DATA_BLOCK "DB09_TablePos"   // DB9
{ S7_Optimized_Access := 'FALSE' }
AUTHOR : Robopac
VERSION : 0.0
// stored: AutoNumber false, IsOnlyStoredInLoadMemory false, IsWriteProtectedInAS false
   VAR RETAIN
      dbx0_0 : Bool := FALSE;
      dbx0_1 : Bool := FALSE;
      dbx0_2 : Bool := TRUE;
      dbx0_3 : Bool := FALSE;
      dbx0_4 : Bool := FALSE;
      dbx0_5 : Bool := FALSE;
      dbx0_6 : Bool := FALSE;
      dbx0_7 : Bool := FALSE;
      dbx1_0 : Bool := FALSE;   // Table rotation axis movement forward
      dbx1_1 : Bool := FALSE;   // Table rotation axis movement backward
      dbx1_2 : Bool := FALSE;   // Table rotation axis movement inside low speed area
      dbx1_3 : Bool := FALSE;   // Table rotation axis movement low speed
      dbx1_4 : Bool := FALSE;   // Table rotation forward
      dbx1_5 : Bool := FALSE;   // Table rotation backward
      dbx1_6 : Bool := TRUE;
      dbx1_7 : Bool := FALSE;
      dbx2_0 : Bool := FALSE;
      dbx2_1 : Bool := FALSE;
      dbx2_2 : Bool := FALSE;
      dbx2_3 : Bool := FALSE;
      dbx2_4 : Bool := FALSE;
      dbx2_5 : Bool := FALSE;
      dbx2_6 : Bool := FALSE;
      dbx2_7 : Bool := FALSE;
      dbx3_0 : Bool := FALSE;   // Table rotation: Support for encoder running control
      dbx3_1 : Bool := FALSE;   // Table rotation: Support for encoder running control alarm
      dbx3_2 : Bool := FALSE;
      dbx3_3 : Bool := FALSE;
      dbx3_4 : Bool := FALSE;
      dbx3_5 : Bool := FALSE;
      dbx3_6 : Bool := FALSE;
      dbx3_7 : Bool := FALSE;
      dbx4_0 : Bool := FALSE;
      dbx4_1 : Bool := FALSE;
      dbx4_2 : Bool := FALSE;
      dbx4_3 : Bool := FALSE;
      dbx4_4 : Bool := FALSE;
      dbx4_5 : Bool := FALSE;
      dbx4_6 : Bool := FALSE;
      dbx4_7 : Bool := FALSE;
      dbx5_0 : Bool := FALSE;
      dbx5_1 : Bool := FALSE;
      dbx5_2 : Bool := FALSE;
      dbx5_3 : Bool := FALSE;
      dbw6 : Int := 5;   // Table rotation: Support for movement speed
      dbw8 : Int := 0;   // Table rotation: Support for movement deceleration
      dbw10 : Int := 5;   // Table rotation inverter: Support for speed selection
      dbw12 : Int := 10199;
      dbw14 : Int := 2340;
      dbw16 : Int := 0;
      dbw18 : Int := 0;
      dbw20 : Int := 0;
      dbw22 : Int := 0;
      dbw24 : Int := 0;
      dbw26 : Int := 0;
      dbw28 : Int := 0;
      dbd30 : DInt := -15;   // Table rotation position: Pulse
      dbw34 : Int := -8;   // Table position
      dbw36 : Int := 0;   // Table rotation position: Table maximum position
      dbw38 : Int := 0;   // Table rotation position: Deceleration position
      dbw40 : Int := 0;   // Table rotation position: Deceleration position
      dbd42 : DInt := -15;   // Support for encoder table rotation running control
      dbw46 : Int := 20;   // Support for encoder table rotation running control
      dbw48 : Int := -8;   // Table position according to offset
      dbw50 : Int := 0;
      dbw52 : Int := 0;
      dbw54 : Int := 0;
      dbw56 : Int := 0;
      dbw58 : Int := 0;
      dbw60 : Int := 0;
      dbw62 : Int := 0;
      dbw64 : Int := 0;
      dbw66 : Int := 0;
      dbw68 : Int := 0;
      dbw70 : Int := 0;
      Req1_Dest : Int := 0;   // Positioning request 1: Destination position
      Req2_Dest : Int := 0;   // Positioning request 2: Destination position
      Req3_Dest : Int := 0;   // Positioning request 3: Destination position
      Req4_Dest : Int := 0;   // Positioning request 4: Destination position
      Req1_Fwd : Bool := FALSE;   // Positioning request 1: Axis forward
      Req1_Bkw : Bool := FALSE;   // Positioning request 1: Axis backward
      Req1_Slow : Bool := FALSE;   // Positioning request 1: Axis slow speed
      Req1_Pos : Bool := FALSE;   // Positioning request 1: Axis in position
      Req2_Fwd : Bool := FALSE;   // Positioning request 2: Axis forward
      Req2_Bkw : Bool := FALSE;   // Positioning request 2: Axis backward
      Req2_Slow : Bool := FALSE;   // Positioning request 2: Axis slow speed
      Req2_Pos : Bool := FALSE;   // Positioning request 2: Axis in position
      Req3_Fwd : Bool := FALSE;   // Positioning request 3: Axis forward
      Req3_Bkw : Bool := FALSE;   // Positioning request 3: Axis backward
      Req3_Slow : Bool := FALSE;   // Positioning request 3: Axis slow speed
      Req3_Pos : Bool := FALSE;   // Positioning request 3: Axis in position
      Req4_Fwd : Bool := FALSE;   // Positioning request 4: Axis forward
      Req4_Bkw : Bool := FALSE;   // Positioning request 4: Axis backward
      Req4_Slow : Bool := FALSE;   // Positioning request 4: Axis slow speed
      Req4_Pos : Bool := FALSE;   // Positioning request 4: Axis in position
      Req5_Dest : Int := 0;   // Positioning request 4: Destination position
      Req6_Dest : Int := 0;   // Positioning request 4: Destination position
      Req7_Dest : Int := 0;   // Positioning request 4: Destination position
      Req8_Dest : Int := 0;   // Positioning request 4: Destination position
      Req5_Fwd : Bool := FALSE;   // Positioning request 5: Axis forward
      Req5_Bkw : Bool := FALSE;   // Positioning request 5: Axis backward
      Req5_Slow : Bool := FALSE;   // Positioning request 5: Axis slow speed
      Req5_Pos : Bool := FALSE;   // Positioning request 5: Axis in position
      Req6_Fwd : Bool := FALSE;   // Positioning request 6: Axis forward
      Req6_Bkw : Bool := FALSE;   // Positioning request 6: Axis backward
      Req6_Slow : Bool := FALSE;   // Positioning request 6: Axis slow speed
      Req6_Pos : Bool := FALSE;   // Positioning request 6: Axis in position
      Req7_Fwd : Bool := FALSE;   // Positioning request 7: Axis forward
      Req7_Bkw : Bool := FALSE;   // Positioning request 7: Axis backward
      Req7_Slow : Bool := FALSE;   // Positioning request 7: Axis slow speed
      Req7_Pos : Bool := FALSE;   // Positioning request 7: Axis in position
      Req8_Fwd : Bool := FALSE;   // Positioning request 8: Axis forward
      Req8_Bkw : Bool := FALSE;   // Positioning request 8: Axis backward
      Req8_Slow : Bool := FALSE;   // Positioning request 8: Axis slow speed
      Req8_Pos : Bool := FALSE;   // Positioning request 8: Axis in position
      dbw92 : Int := 0;
      dbw94 : Int := 0;
      dbw96 : Int := 0;
      dbw98 : Int := 0;
   END_VAR
BEGIN
END_DATA_BLOCK

DATA_BLOCK "DB100_Display"   // DB100
{ S7_Optimized_Access := 'FALSE' }
VERSION : 0.1
// stored: AutoNumber false, IsOnlyStoredInLoadMemory false, IsWriteProtectedInAS false
   VAR RETAIN
      CELLA : Int := 15;   // CELLA (rosa)
      SETPOINT : UInt := 20;   // SETPOINT (rosso)
      PROP : Int := 0;   // PROPORZIONALE (verde)
      "INT" : Int := 0;   // INTEGRALE (giallo)
      FREQ_TIRO : Int := 0;   // U241
      FREQ_PRES : Int := 0;   // U261
   END_VAR
BEGIN
END_DATA_BLOCK

DATA_BLOCK "DB10_ExtConveyors"   // DB10
{ S7_Optimized_Access := 'FALSE' }
VERSION : 0.1
// stored: AutoNumber false, IsOnlyStoredInLoadMemory false, IsWriteProtectedInAS false
   VAR RETAIN
      V1000_0 : Bool := FALSE;
      V1000_1 : Bool := FALSE;
      V1000_2 : Bool := FALSE;
      V1000_3 : Bool := FALSE;
      V1000_4 : Bool := FALSE;
      V1000_5 : Bool := FALSE;
      V1000_6 : Bool := FALSE;
      V1000_7 : Bool := FALSE;
      V1001_0 : Bool := FALSE;
      V1001_1 : Bool := FALSE;
      V1001_2 : Bool := FALSE;
      V1001_3 : Bool := FALSE;
      V1001_4 : Bool := FALSE;
      V1001_5 : Bool := FALSE;
      V1001_6 : Bool := FALSE;
      V1001_7 : Bool := FALSE;
      Out_ConvPos1 : Bool := FALSE;   // Conveyor pos1 motor
      Out_ConvPos2 : Bool := FALSE;   // Conveyor pos2 motor
      Out_ConvPos3 : Bool := FALSE;   // Conveyor pos3 motor
      Out_ConvPos4 : Bool := FALSE;   // Conveyor pos4 motor
      Out_ConvPos5 : Bool := FALSE;   // Conveyor pos5 motor
      Out_ConvPos6 : Bool := FALSE;   // Conveyor pos6 motor
      Out_ConvPos7 : Bool := FALSE;   // Conveyor pos7 motor
      Out_ConvPos8 : Bool := FALSE;   // Conveyor pos8 motor
      Out_ConvPos1Rev : Bool := FALSE;   // Conveyor pos1 motor reverse
      Out_ConvPos2Rev : Bool := FALSE;   // Conveyor pos2 motor reverse
      Out_ConvPos3Rev : Bool := FALSE;   // Conveyor pos3 motor reverse
      Out_ConvPos4Rev : Bool := FALSE;   // Conveyor pos4 motor reverse
      V1003_4 : Bool := FALSE;
      V1003_5 : Bool := FALSE;
      V1003_6 : Bool := FALSE;
      V1003_7 : Bool := FALSE;
      VW1004 : Int := 0;
      Out_ConvPos1X2 : Bool := FALSE;   // Conveyor pos1 motor speed selection X2
      Out_ConvPos2X2 : Bool := FALSE;   // Conveyor pos2 motor speed selection X2
      Out_ConvPos3X2 : Bool := FALSE;   // Conveyor pos3 motor speed selection X2
      Out_ConvPos4X2 : Bool := FALSE;   // Conveyor pos4 motor speed selection X2
      V1006_4 : Bool := FALSE;
      V1006_5 : Bool := FALSE;
      V1006_6 : Bool := FALSE;
      V1006_7 : Bool := FALSE;
      Out_ConvPos2Upw : Bool := FALSE;   // Conveyor pos2 motor upward
      Out_ConvPos2Downw : Bool := FALSE;   // Conveyor pos2 downstroke valve command
      In_ConvPos2Up : Bool := TRUE;   // Conveyor pos2 up photocell NC
      In_ConvPos2Down : Bool := TRUE;   // Conveyor pos2 down photocell NC
      In_ConvPos2ExUp : Bool := TRUE;   // Conveyor pos2 up extrastroke switch NC
      In_ConvPos2Safety : Bool := TRUE;   // Conveyor pos2 down foot safety switch NC
      V1007_6 : Bool := FALSE;
      V1007_7 : Bool := FALSE;
   END_VAR
BEGIN
END_DATA_BLOCK

DATA_BLOCK "DB13_TableFaseControl"   // DB13
{ S7_Optimized_Access := 'FALSE' }
VERSION : 0.1
// stored: AutoNumber false, IsOnlyStoredInLoadMemory false, IsWriteProtectedInAS false
   VAR RETAIN
      load : Bool := TRUE;
      cm : Bool := TRUE;
      unload : Bool := TRUE;
      hysteresis : Int := 100;
   END_VAR
BEGIN
END_DATA_BLOCK

DATA_BLOCK "DB14_CutWireControl"   // DB14
{ S7_Optimized_Access := 'FALSE' }
VERSION : 0.1
// stored: AutoNumber false, IsOnlyStoredInLoadMemory false, IsWriteProtectedInAS false
   VAR RETAIN
      clean : Time := T#0MS;
      check : Time := T#0MS;
   END_VAR
BEGIN
END_DATA_BLOCK

DATA_BLOCK "DB18_TableSpeed"   // DB18
{ S7_Optimized_Access := 'FALSE' }
VERSION : 0.1
// stored: AutoNumber false, IsOnlyStoredInLoadMemory false, IsWriteProtectedInAS false
   VAR RETAIN
      spare0 : Int := 0;
      spare1 : Int := 0;
      spare2 : Int := 0;
      spare3 : Int := 0;
      spare4 : Int := 0;
      spare5 : Int := 0;
      spare6 : Int := 0;
      spare7 : Int := 0;
      DBD16 : Real := 0.0;   // Actual speed in degrees per second (split before use)
      DBD20 : Real := 90.0;   // Low speed in degrees per second (split before use)
      DBD24 : Real := 900.0;   // High speed in degrees per second (split before use)
      spare14 : Int := 0;
      DBW30 : Int := 0;   // Degrees to reach minimum speed from maximum speed
      spare16 : Int := 0;
      DBW34 : Int := 50;
   END_VAR
BEGIN
END_DATA_BLOCK

DATA_BLOCK "DB20_DisplaySysdata"   // DB20
{ S7_Optimized_Access := 'FALSE' }
AUTHOR : Robopac
VERSION : 0.0
// stored: AutoNumber false, IsOnlyStoredInLoadMemory false, IsWriteProtectedInAS false
   VAR RETAIN
      dbd0 : DInt := 238;   // Step for encoder spool carriage movement (mm/100) (Display-Sysadata)
      dbw4 : Int := 6;   // Histeresys for spool carriage positioning (mm) (Display-Sysdata)
      dbw6 : Int := 50;   // Deceleration for spool carriage positioning (mm) (Display-Sysdata)
      dbw8 : Int := 50;   // Low speed for spool carriage movement (%) (Display-Sysdata)
      dbw10 : Int := 100;   // High speed for spool carriage movement (%) (Display-Sysdata)
      dbw12 : Int := 430;   // Spool height (mm) (Display-Sysdata)
      dbw14 : Int := 0;   // Spool carriage down position (mm) (Display-Sysadata)
      dbw16 : Int := 100;   // First step speed for spool carriage movement (%) (Display-Sysadata)
      dbw18 : Int := 240;   // Offset for ftc pallet height (mm) (Display-Sysdata)
      dbw20 : Int := 180;   // Pressure plate height (mm) (Display-Sysdata)
      dbw22 : Int := 7;   // Distance lifter up - conveyor (mm) (Display-Sysdata)
      dbw24 : Int := 0;   // Spool carriage height for film broken cycle (mm) (Display-Sysdata)
      dbw26 : Int := 50;   // Low speed angle to stop rotation (Display-Sysdata)
      dbw28 : Int := 1000;   // Jog1 speed for fast prestretch rool (Display-Sysadata)
      dbw30 : Int := 45;   // Offset for SCSP/2 (Display-Sysadata)
      dbw32 : Int := 78;
      dbw34 : Int := 1100;   // Arm rotation motor and gearbox type (Display-Sysdata)
      dbw36 : Int := 0;   // Delay for test cycle (Display-Sysdata)
      dbx38_0 : Bool := FALSE;   // Film ended or broken cycle included/excluded(1) (Display-Sysdata)
      dbx38_1 : Bool := FALSE;   // Conveyor encoder alarm included(0)/excluded (Display-Sysdata)
      dbx38_2 : Bool := FALSE;   // Test cycle included(1)/excluded (Display-Sysdata)
      dbx38_3 : Bool := FALSE;   // Top film ended or broken included(0)/excluded (Display-Sysdata)
      dbx38_4 : Bool := TRUE;   // Pallet height with pressure plate priority (Display-Sysdata)
      dbx38_5 : Bool := TRUE;   // Spool carriage upward during arm deceleration excluded/included(1) (Display-Sys
      dbx38_6 : Bool := FALSE;   // Pressure plate upward before(0)/after cut cycle (Display-Sysdata)
      dbx38_7 : Bool := FALSE;   // Bit stop pallet infeed (Display-Sysdata)
      dbx39_0 : Bool := FALSE;   // Timeout included/excluded(1) (Display-Sysdata)
      dbx39_1 : Bool := FALSE;   // Reverse cycle request from hmi (Display-Main page)
      dbx39_2 : Bool := FALSE;
      dbx39_3 : Bool := FALSE;
      dbx39_4 : Bool := FALSE;
      dbx39_5 : Bool := FALSE;
      dbx39_6 : Bool := TRUE;   // Top fast cycle
      dbx39_7 : Bool := FALSE;
      dbw40 : Int := 65;   // Spool carriage upward during arm deceleration (mm) (Display-Sysdata)
      dbw42 : Int := 1360;   // Step for infeed conveyor encoder (mm/100) (Display-Sysdata)
      dbw44 : Int := -210;   // Pulse offset for rotation encoder (Display-Sysdata)
      dbw46 : Int := 0;   // Pallet lenght for small pallet (Display-Sysdata)
      dbw48 : Int := 0;   // Decentering for pallet positioning (Display-Sysdata)
      dbw50 : Int := 500;   // Quote for airblower on (mm) (Display-Sysdata)
      dbw52 : Int := 0;   // Spool carriage up to cover film tail (Display-Sysdata)
      dbw54 : Int := 3000;   // Cutting time (Display-Sysdata)
      dbw56 : Int := 1500;   // MAX TIRO SU CELLA (kg) [ex SysdataTempoTwist]
      dbw58 : Int := 2400;   // Delay to open clamp (Display-Sysdata)
      dbw60 : Int := 0;   // Table rotation clampcut phase (°) (Display-Sysdata)
      dbw62 : Int := 200;   // Quote to open clamp (Display-Sysdata)
      dbw64 : Int := 0;   // Step for top carriage forward/backward (mm/100) (Display-Sysdata)
      dbw66 : Int := 1000;   // Step for top carriage upward/downward (mm/100) (Display-Sysdata)
      dbw68 : Int := 600;   // Deceleration for top carriage forward/backward (Display-Sysdata)
      dbw70 : Int := 1500;   // Top carriage up position (Display-Sysdata)
      dbw72 : Int := 0;   // Spool carriage position for top cycle (Display-Sysdata)
      dbw74 : Int := 0;   // Delay for spool carriage downward during top cycle (Display-Sysdata)
      dbw76 : Int := 0;   // Tabke rotation load phase (°) (Display-Sysdata)
      dbw78 : Int := 0;   // Table rotation unload phase (°) (Display-Sysdata)
      dbd80 : DInt := 5627;   // Step for encoder table rotation movement (°/p) (Display-Sysdata)
      dbw84 : Int := 18;   // Histeresys for table rotation positioning (°) (Display-Sysdata)
      dbw86 : Int := 2100;   // Deceleration for table rotation positioning (Hz/sec) (Display-Sysdata)
      dbw88 : Int := 10;   // Low speed for table rotation movement (%) (Display-Sysdata)
      dbw90 : Int := 100;   // High speed for table rotation movement (%) (Display-Sysdata)
      dbw92 : Int := 1800;   // Delay to stop top carriage forward for top film broken
      dbw94 : Int := 1000;   // Delay for top pallet height reading photocell (fast cycle)
      dbw96 : Int := 60;
      dbw98 : Int := 20;
   END_VAR
BEGIN
END_DATA_BLOCK

DATA_BLOCK "DB215_ProgramData"   // DB215
TITLE = Program Data
{ S7_Optimized_Access := 'FALSE' }
VERSION : 0.1
// stored: AutoNumber false, IsOnlyStoredInLoadMemory false, IsWriteProtectedInAS false
   VAR RETAIN
      State_Initialization : UInt := 0;
      State_Setup : UInt := 0;
      InverterFault : Bool := FALSE;   // Inverter Fault (F) - Anomalia
      InverterAlarm : Bool := FALSE;   // Inverter Alarm (A) - Avviso
      Keylock : Bool := FALSE;   // Blocco tasti per utente
      ActiveRecipeMLC : Bool := FALSE;   // Multi-Level Control per la ricetta attiva
      Keylock2 : Bool := FALSE;   // Blocco tasti (StateAuto opp. blocco)
      RecipeModified : Bool := FALSE;
      RecipeSave : Bool := FALSE;
      LoadCellConst : Bool := TRUE;   // valore cella costante
      spare_5 : Bool := FALSE;
      spare_6 : Bool := FALSE;
      spare_7 : Bool := FALSE;
      spare_8 : Bool := FALSE;
      spare_9 : Bool := FALSE;
      spare_10 : Bool := FALSE;
      spare_11 : Bool := FALSE;
      spare_12 : Bool := FALSE;
      Offset_Pulses : Int := 0;   // NOT_USED
      Altimeter_Pulses : Int := 442;
      PhotDelay_Pulses : Int := 40;
      Reinforce_Pulses : Int := 0;
      TopFall_Pulses : Int := 134;
      ManRotStep : UInt := 0;
      RotSpeed : Int := 1770;
      CarSpeedUp : Int := 1396;
      CarSpeedDw : Int := 1396;
      Offset_cella : Int := 240;
      EncCarrDir : Int := -1;   // Direzione petalo carrello (1=av;-1=ind)
      EncCarrMax : Int := 603;   // Max altezza carrello (encoder)
      TiroObiettivo : UInt := 0;   // Tiro obiettivo (da chiamata FC300)
      ContaImpulsi : Int := 0;   // Contatore impulsi 20ms (OB30)
      MLC_HeightPulses : Int := 0;   // MLC_Height_Pulses
      MLC_Rounds : Int := 0;   // MLC_rounds
      LoadCellVal_1 : Int := 227;   // valore cella 1
      LoadCellVal_2 : Int := 227;   // valore cella 2
      PropArmMax : Int := 0;   // Costante proporzionalità corrisp. max freq. braccio
      PropCarrMax : Int := 0;   // Costante proporzionalità corrisp. max freq. carrello
      ValOffsetCella : Int := 10;   // Valore per offset cella durante il reset
      RoundTime : UInt := 4000;
      LastRoundTime : UInt := 2000;
      ReinforceTime : UInt := 0;   // [NOT USED]
      pTiro : Array[0..10] of UInt;
      iTiro : Array[0..10] of UInt;
   END_VAR
BEGIN
   pTiro[0] := 70;
   pTiro[1] := 60;
   pTiro[2] := 50;
   pTiro[3] := 45;
   pTiro[4] := 40;
   pTiro[5] := 35;
   pTiro[6] := 30;
   pTiro[7] := 25;
   pTiro[8..10] := 20;
   iTiro[0] := 70;
   iTiro[1] := 60;
   iTiro[2] := 50;
   iTiro[3] := 45;
   iTiro[4] := 40;
   iTiro[5] := 35;
   iTiro[6] := 30;
   iTiro[7] := 25;
   iTiro[8..10] := 20;
END_DATA_BLOCK

DATA_BLOCK "DB21_DisplayGeneralData"   // DB21
{ S7_Optimized_Access := 'FALSE' }
AUTHOR : Robopac
VERSION : 0.0
// stored: AutoNumber false, IsOnlyStoredInLoadMemory false, IsWriteProtectedInAS false
   VAR RETAIN
      dbx0_0 : Bool := TRUE;   // Welder unit included(1)/excluded (Display-General Data)
      dbx0_1 : Bool := FALSE;   // Machine included(1)/excluded (Display-General Data)
      dbx0_2 : Bool := TRUE;   // Pallet load/unload included(1)/excluded (Display-Sysdata)
      dbx0_3 : Bool := TRUE;   // Load pallet with forklift selection by display (Display-Sysdata)
      dbx0_4 : Bool := TRUE;   // Unload pallet with forklift selection by display (Display-Sysdata)
      dbx0_5 : Bool := FALSE;
      dbx0_6 : Bool := TRUE;
      dbx0_7 : Bool := FALSE;
      dbb1 : Byte := 16#00;
      dbw2 : Int := 3;   // PLC SW major release
      dbw4 : Int := 0;   // PLC SW minor release
      dbw6 : Int := 90;   // Spool carriage upward for spring clamp at begin cycle (Display-General Data)
      dbw8 : Int := 0;   // Spool carriage downward for film tail at the cycle begin (Display-General Data)
      dbw10 : Int := 2;   // Film thickness (Display-General Data)
      dbw12 : Int := 700;   // Welding time (Display-General Data)
      dbw14 : Int := 0;   // Low speed for Helix conveyor movement (%) (Display-Sysdata)
      dbw16 : Int := 0;   // High speed for Helix conveyor movement (%) (Display-Sysdata)
      dbw18 : Int := 500;   // Delay on pallet positioning (Display-General Data)
      dbw20 : Int := 10000;   // Delay for load/unload pallet simultaneously (Display-General Data)
      dbw22 : Int := 100;   // Deceleration for pallet positioning (Display-General Data)
      dbw24 : Int := 1;   // Time for pallet load with forklift
      dbw26 : Int := 0;   // Override for ring movement in manul mode (Display-General Data)
      dbw28 : Int := 100;   // TIMER CICLO FIERA (attesa tra cicli successivi)
      dbw30 : Int := 0;   // Film prestretch for film prestretch test cycle (Display-General Data)
      dbw32 : Int := 0;   // Film prestretch increase for film prestretch test (Display-General Data)
      dbw34 : Int := 0;   // Film supplied every revolution for film prestretch test (Display-General Data)
      dbw36 : Int := 0;   // Time for spool carriage upward for table cycle (Display-Sysdata)
      dbw38 : Int := 2000;   // Time for spool carriage upward for table cycle (Display-Sysdata)
      dbw40 : Int := 15000;   // Time load with forklift
      dbw42 : Int := 10000;   // Time unload with forklift
   END_VAR
BEGIN
END_DATA_BLOCK

DATA_BLOCK "DB22_DisplayData"   // DB22
{ S7_Optimized_Access := 'FALSE' }
AUTHOR : Robopac
VERSION : 0.0
// stored: AutoNumber false, IsOnlyStoredInLoadMemory false, IsWriteProtectedInAS false
   VAR RETAIN
      dbx0_0 : Bool := FALSE;   // Technoplat manual(Display): Table rotation forward
      dbx0_1 : Bool := FALSE;   // Technoplat manual(Display): Spool carriage upward
      dbx0_2 : Bool := FALSE;   // Technoplat manual(Display): Spool carriage downward
      dbx0_3 : Bool := FALSE;   // Technoplat manual(Display): Pressure plate upward/downward
      dbx0_4 : Bool := FALSE;   // Technoplat manual(Display): Pallet lifter upward/downward
      dbx0_5 : Bool := FALSE;   // Technoplat manual(Display): Rope unit open/close
      dbx0_6 : Bool := FALSE;   // Technoplat manual(Display): Prestretch
      dbx0_7 : Bool := FALSE;   // Technoplat manual(Display): Spool carriage to film broken position
      dbx1_0 : Bool := FALSE;   // Clamp manual(Display): Clamp upward/downward
      dbx1_1 : Bool := FALSE;   // Clamp manual(Display): Welder unit upward/downward
      dbx1_2 : Bool := FALSE;   // Clamp manual(Display): Welder contrast upward/downward
      dbx1_3 : Bool := FALSE;   // Clamp manual(Display): Clamp carriage forward/backward
      dbx1_4 : Bool := FALSE;   // Clamp manual(Display): Clamp open/close
      dbx1_5 : Bool := FALSE;   // Clamp manual(Display): Cut and welder arm forward/backward
      dbx1_6 : Bool := FALSE;   // Clamp manual(Display): Welder unit forward/backward
      dbx1_7 : Bool := FALSE;   // Clamp manual(Display):
      dbx2_0 : Bool := FALSE;   // Top manual(Display): Top carriage upward
      dbx2_1 : Bool := FALSE;   // Top manual(Display): Top carriage downward
      dbx2_2 : Bool := FALSE;   // Top manual(Display): Top carriage forward
      dbx2_3 : Bool := FALSE;   // Top manual(Display): Top carriage backward
      dbx2_4 : Bool := FALSE;   // Top manual(Display): Opening/closing clamp to pull top film
      dbx2_5 : Bool := FALSE;   // Top manual(Display): Opening/closing clamp to block top film
      dbx2_6 : Bool := FALSE;   // Top manual(Display): Top film cutter forward/backward
      dbx2_7 : Bool := FALSE;   // Top manual(Display): Arm rotation to phase 2 sensor for top
      dbx3_0 : Bool := FALSE;   // Technoplat manual (Display): Rotation to unload
      dbx3_1 : Bool := FALSE;   // Technoplat manual (Display): Rotation to 0
      dbx3_2 : Bool := FALSE;   // Technoplat manual (Display): Rotation to load
      dbx3_3 : Bool := FALSE;
      dbx3_4 : Bool := FALSE;   // Technoplat manual(Display): Rope unit lower open/close
      dbx3_5 : Bool := FALSE;
      dbx3_6 : Bool := FALSE;
      dbx3_7 : Bool := FALSE;
      dbx4_0 : Bool := FALSE;   // Conveyor manual(Display): CMD PRESSED
      dbx4_1 : Bool := FALSE;   // Conveyor manual(Display): Load CM [p18]
      dbx4_2 : Bool := FALSE;   // Conveyor manual(Display): Unload CM [p18]
      dbx4_3 : Bool := FALSE;   // Conveyor manual(Display): RESET ENCODER
      dbx4_4 : Bool := FALSE;   // Conveyor manual(Display): Load CM [Sysdata]
      dbx4_5 : Bool := FALSE;   // Conveyor manual(Display): [not used]
      dbx4_6 : Bool := FALSE;   // Conveyor manual(Display): CM backward slow
      dbx4_7 : Bool := FALSE;   // Conveyor manual(Display): CM forward slow
      dbb5 : Byte := 16#09;   // Conveyor manual operation
      dbx6_0 : Bool := FALSE;   // Manual Signal(Display): Pallet ready in infeed (Input)
      dbx6_1 : Bool := FALSE;   // Manual Signal(Display): Ready to receive pallet infeed (Output)
      dbx6_2 : Bool := FALSE;   // Manual Signal(Display): End of transfer pallet infeed (Output)
      dbx6_3 : Bool := FALSE;   // Manual Signal(Display): Pallet ready in outfeed (Output)
      dbx6_4 : Bool := FALSE;   // Manual Signal(Display): Ready to receive pallet outfeed (Input)
      dbx6_5 : Bool := FALSE;   // Manual Signal(Display): End of transfer pallet outfeed (Input)
      dbx6_6 : Bool := FALSE;   // Manual Signal(Display): Start wrapping signal (Input)
      dbx6_7 : Bool := FALSE;   // Manual Signal(Display): Customer conveyor stopped signal (Input)
      dbx7_0 : Bool := FALSE;   // Manual Signal(Display): Machine in position signal (Output)
      dbx7_1 : Bool := FALSE;   // Manual Signal(Display): Wrapp ended signal (Output)
      dbx7_2 : Bool := FALSE;   // Manual Signal(Display): Pallet in position for label
      dbx7_3 : Bool := TRUE;   // Manual Signal(Display): Label arm in position for pallet transfer
      dbx7_4 : Bool := FALSE;   // Manual Signal(Display): Label cycle ended
      dbx7_5 : Bool := FALSE;   // Manual Signal(Display): Label fault
      dbx7_6 : Bool := FALSE;
      dbx7_7 : Bool := FALSE;
      dbw8 : Int := 0;
      dbw10 : Int := 0;
      dbw12 : Int := 0;
      dbx14_0 : Bool := FALSE;   // Technoplat manual(Program): Table rotation forward
      dbx14_1 : Bool := FALSE;   // Technoplat manual(Program): Spool carriage upward
      dbx14_2 : Bool := FALSE;   // Technoplat manual(Program): Spool carriage downward
      dbx14_3 : Bool := FALSE;   // Technoplat manual(Program): Pressure plate downward
      dbx14_4 : Bool := FALSE;   // Technoplat manual(Program): Pressure plate upward
      dbx14_5 : Bool := FALSE;   // Technoplat manual(Program): Pallet lifter upward
      dbx14_6 : Bool := FALSE;   // Technoplat manual(Program): Pallet lifter downward
      dbx14_7 : Bool := FALSE;   // Technoplat manual(Program): Rope unit closing
      dbx15_0 : Bool := FALSE;   // Technoplat manual(Program): Rope unit opening
      dbx15_1 : Bool := FALSE;   // Technoplat manual(Program): Prestretch
      dbx15_2 : Bool := FALSE;   // Technoplat manual(Program): Spool carriage to film broken position
      dbx15_3 : Bool := FALSE;   // Technoplat manual(Program): Rope unit Lower closing
      dbx15_4 : Bool := FALSE;   // Technoplat manual(Program): Rope unit Lower opening
      dbx15_5 : Bool := FALSE;   // Technoplat manual(Program): CM Backward slow
      dbx15_6 : Bool := FALSE;   // Technoplat manual(Program): CM Forward slow
      dbx15_7 : Bool := FALSE;   // Technoplat manual(Program):
      dbx16_0 : Bool := FALSE;   // Clamp manual(Program): Clamp upward
      dbx16_1 : Bool := FALSE;   // Clamp manual(Program): Clamp downward
      dbx16_2 : Bool := FALSE;   // Clamp manual(Program): Welder unit upward
      dbx16_3 : Bool := FALSE;   // Clamp manual(Program): Welder unit downward
      dbx16_4 : Bool := FALSE;   // Clamp manual(Program): Welder contrast upward
      dbx16_5 : Bool := FALSE;   // Clamp manual(Program): Welder contrast downward
      dbx16_6 : Bool := FALSE;   // Clamp manual(Program): Clamp carriage forward
      dbx16_7 : Bool := FALSE;   // Clamp manual(Program): Clamp carriage backward
      dbx17_0 : Bool := FALSE;   // Clamp manual(Program): Clamp open
      dbx17_1 : Bool := FALSE;   // Clamp manual(Program): Clamp close
      dbx17_2 : Bool := FALSE;   // Clamp manual(Program): Cut and welder arm forward
      dbx17_3 : Bool := FALSE;   // Clamp manual(Program): Cut and welder arm backward
      dbx17_4 : Bool := FALSE;   // Clamp manual(Program): Welder unit forward
      dbx17_5 : Bool := FALSE;   // Clamp manual(Program): Welder unit backward
      dbx17_6 : Bool := FALSE;   // Clamp manual(Program):
      dbx17_7 : Bool := FALSE;   // Clamp manual(Program):
      dbx18_0 : Bool := FALSE;   // Top manual(Program): Top carriage upward
      dbx18_1 : Bool := FALSE;   // Top manual(Program): Top carriage downward
      dbx18_2 : Bool := FALSE;   // Top manual(Program): Top carriage forward
      dbx18_3 : Bool := FALSE;   // Top manual(Program): Top carriage backward
      dbx18_4 : Bool := FALSE;   // Top manual(Program): Opening clamp to pull top film
      dbx18_5 : Bool := FALSE;   // Top manual(Program): Closing clamp to pull top film
      dbx18_6 : Bool := FALSE;   // Top manual(Program): Opening clamp to block top film
      dbx18_7 : Bool := FALSE;   // Top manual(Program): Closing clamp to block top film
      dbx19_0 : Bool := FALSE;   // Top manual(Program): Top film cutter forward/backward
      dbx19_1 : Bool := FALSE;   // Top manual(Program): Arm rotation to phase 2 sensor for top
      dbx19_2 : Bool := FALSE;   // Technoplat manual(Program): Rotation to unload
      dbx19_3 : Bool := FALSE;   // Technoplat manual(Program): Rotation to 0
      dbx19_4 : Bool := FALSE;   // Technoplat manual(Program): Rotation to load
      dbx19_5 : Bool := FALSE;   // Top manual(Program):
      dbx19_6 : Bool := FALSE;   // Top manual(Program):
      dbx19_7 : Bool := FALSE;   // Top manual(Program):
      dbx20_0 : Bool := FALSE;   // Conveyor manual(Program): Load CM
      dbx20_1 : Bool := FALSE;   // Conveyor manual(Program): Unload CM
      dbx20_2 : Bool := FALSE;   // Conveyor manual(Program): CM backward
      dbx20_3 : Bool := FALSE;   // Conveyor manual(Program): Pos.1
      dbx20_4 : Bool := FALSE;   // Conveyor manual(Program): Pos.2
      dbx20_5 : Bool := FALSE;   // Conveyor manual(Program): Pos.3
      dbx20_6 : Bool := FALSE;   // Conveyor manual(Program): Pos.4
      dbx20_7 : Bool := FALSE;   // Conveyor manual(Program): Pos.5
      dbx21_0 : Bool := FALSE;   // Conveyor manual(Program): Pos.6
      dbx21_1 : Bool := FALSE;   // Conveyor manual(Program): Pos.7
      dbx21_2 : Bool := FALSE;   // Conveyor manual(Program): Pos.8
      dbx21_3 : Bool := FALSE;   // Conveyor manual(Program):
      dbx21_4 : Bool := FALSE;   // Conveyor manual(Program):
      dbx21_5 : Bool := FALSE;   // Conveyor manual(Program):
      dbx21_6 : Bool := FALSE;   // Conveyor manual(Program):
      dbx21_7 : Bool := FALSE;   // Conveyor manual(Program):
      dbx22_0 : Bool := FALSE;   // Manual Signal(Program): Pallet ready in infeed (Input)
      dbx22_1 : Bool := FALSE;   // Manual Signal(Program): Ready to receive pallet infeed (Output)
      dbx22_2 : Bool := FALSE;   // Manual Signal(Program): End of transfer pallet infeed (Output)
      dbx22_3 : Bool := FALSE;   // Manual Signal(Program): Pallet ready in outfeed (Output)
      dbx22_4 : Bool := FALSE;   // Manual Signal(Program): Ready to receive pallet outfeed (Input)
      dbx22_5 : Bool := FALSE;   // Manual Signal(Program): End of transfer pallet outfeed (Input)
      dbx22_6 : Bool := FALSE;   // Manual Signal(Program): Start wrapping (Input)
      dbx22_7 : Bool := FALSE;   // Manual Signal(Program): Customer conveyor stopped (Input)
      dbx23_0 : Bool := FALSE;   // Manual Signal(Program): Machine in position (Output)
      dbx23_1 : Bool := FALSE;   // Manual Signal(Program): Wrapp ended (Output)
      dbx23_2 : Bool := FALSE;   // Manual Signal(Program): Pallet ready for label
      dbx23_3 : Bool := TRUE;   // Manual Signal(Program): Label arm in position for pallet transfer
      dbx23_4 : Bool := FALSE;   // Manual Signal(Program): Label cycle ended
      dbx23_5 : Bool := FALSE;   // Manual Signal(Program): Label fault
      dbx23_6 : Bool := FALSE;
      dbx23_7 : Bool := FALSE;
      dbw24 : Int := 0;
      dbw26 : Int := 0;
      dbw28 : Int := 0;
      dbw30 : Int := 0;
      dbx32_0 : Bool := TRUE;   // Manual(Toggle bit): Pressure plate upward/downward (Technplat)
      dbx32_1 : Bool := TRUE;   // Manual(Toggle bit): Pallet lifter upward/downward (Technplat)
      dbx32_2 : Bool := FALSE;   // Manual(Toggle bit): Clamp upward/downward (Clamp)
      dbx32_3 : Bool := FALSE;   // Manual(Toggle bit): Welder unit upward/downward (Clamp)
      dbx32_4 : Bool := TRUE;   // Manual(Toggle bit): Welder contrast upward/downward (Clamp)
      dbx32_5 : Bool := FALSE;   // Manual(Toggle bit): Rope unit open/close (Technplat)
      dbx32_6 : Bool := FALSE;   // Manual(Toggle bit): Clamp open/close (Clamp)
      dbx32_7 : Bool := FALSE;   // Manual(Toggle bit): Cut and welder arm forward/backward (Clamp)
      dbx33_0 : Bool := TRUE;   // Manual(Toggle bit): Opening/closing clamp to pull top film (Top)
      dbx33_1 : Bool := TRUE;   // Manual(Toggle bit): Opening/closing clamp to block top film (Top)
      dbx33_2 : Bool := TRUE;   // Manual(Toggle bit): Welder unit forward/backward (Clamp)
      dbx33_3 : Bool := FALSE;   // Manual(Toggle bit): Clamp carriage forward/backward (Clamp)
      dbx33_4 : Bool := FALSE;   // Manual(Toggle bit): Rope unit lower open/close (Technplat)
      dbx33_5 : Bool := FALSE;   // Manual(Toggle bit):
      dbx33_6 : Bool := FALSE;   // Manual(Toggle bit):
      dbx33_7 : Bool := FALSE;   // Manual(Toggle bit):
      dbw34 : Int := 0;
      dbw36 : Int := 0;
      dbx38_0 : Bool := FALSE;   // Diagnostic signal conveyor: Pallet ready in infeed (input)
      dbx38_1 : Bool := TRUE;   // Diagnostic signal conveyor: Ready to receive pallet infeed (Output)
      dbx38_2 : Bool := FALSE;   // Diagnostic signal conveyor: End of transfer pallet infeed (Output)
      dbx38_3 : Bool := FALSE;   // Diagnostic signal conveyor: Ready to receive pallet in outfeed (Input)
      dbx38_4 : Bool := FALSE;   // Diagnostic signal conveyor: End of transfer pallet outfeed (Input)
      dbx38_5 : Bool := FALSE;   // Diagnostic signal conveyor: Pallet ready in outfeed (Output)
      dbx38_6 : Bool := FALSE;   // Diagnostic signal conveyor: Start wrapping (Input)
      dbx38_7 : Bool := FALSE;   // Diagnostic signal conveyor: Customer conveyor stopped (Input)
      dbx39_0 : Bool := FALSE;   // Diagnostic signal conveyor: Machine in position (Output)
      dbx39_1 : Bool := FALSE;   // Diagnostic signal conveyor: Wrapp ended (Output)
      dbx39_2 : Bool := FALSE;   // Diagnostic signal conveyor: Pallet ready for label
      dbx39_3 : Bool := TRUE;   // Diagnostic signal conveyor: Label arm in position for pallet transit
      dbx39_4 : Bool := FALSE;   // Diagnostic signal conveyor: Label cycle ended
      dbx39_5 : Bool := FALSE;   // Diagnostic signal conveyor: Label fault
      dbw40 : Int := 1;   // Machine status
      dbd42 : DInt := 4;   // Worked hours
      dbd46 : DInt := 95;   // Partial counter for wrapped pallet
      dbd50 : DInt := 163;   // Counter for wrapped pallet
      dbd54 : DInt := 0;
      dbw58 : Int := 21;   // Seconds for worked hours counter
      dbw60 : Int := 36;   // Minutes for worked hours counter
      dbw62 : Int := 0;   // Arm rotation speed (rpm)
      dbw64 : Int := 0;   // Arm rotation speed (rpm)
      dbw66 : Int := 15;   // Number of revolution done on last pallet
      dbw68 : Int := 777;   // Wrapping cycle time
      dbw70 : Int := 22482;   // Wrapping cycle + pallet transfer time
      dbw72 : Int := 10;   // Pallet per hour (Productivity)
      dbw74 : Int := 0;   // Film weight every wrapping cycle (g*10)
      dbw76 : Int := 0;   // Film force for film weight value
      dbw78 : Int := 0;   // Film prestretch for film weight value
      dbw80 : Int := 0;
      dbw82 : Int := 0;
      dbw84 : Int := 0;
      dbw86 : Int := 0;
      dbw88 : Int := 0;
      dbw90 : Int := 0;
      dbw92 : Int := 0;
      dbw94 : Int := 0;
      dbw96 : Int := 0;
      dbw98 : Int := 0;
   END_VAR
BEGIN
END_DATA_BLOCK

DATA_BLOCK "DB234_Program16"   // DB234
{ S7_Optimized_Access := 'FALSE' }
AUTHOR : Robopac
VERSION : 0.0
// stored: AutoNumber false, IsOnlyStoredInLoadMemory false, IsWriteProtectedInAS false
   VAR RETAIN
      Program16 { S7_SetPoint := 'True'} : "DatiProgramma";
   END_VAR
BEGIN
   Program16.Wrapping := FALSE;
   Program16.TopLenght := 0;
   Program16.TopRelease := 0;
   Program16.TopDown := 0;
   Program16.Top := 0;
   Program16.PressurePTime := 0;
   Program16.LifterTime := 0;
   Program16.RevOverContrast := 0;
   Program16.RopeEndCycle := 16#00;
   Program16.Spare4 := 16#00;
   Program16.RopeTime := 0;
   Program16.RevOverClamp := 0;
   Program16.FilmForceFinalRev := 0;
   Program16.FilmPrestretchFinalRev := 0;
   Program16.ArmSpeed := 0;
   Program16.CarriageDown4Top := 0;
   Program16.TopDownTime := 0;
   Program16.LapsUnderTop := 0;
   Program16.Spare6 := 0;
   Program16.Spare7 := 0;
   Program16.Spare8 := 0;
   Program16.Spare9 := 0;
   Program16.Spare10 := 0;
   Program16.Spare11 := 0;
   Program16.Spare12 := 0;
   Program16.Overlap0_1 := 0;
   Program16.Height1 := 0;
   Program16.Landmark1 := FALSE;
   Program16.Lifter1 := FALSE;
   Program16.SpareBit1H1 := FALSE;
   Program16.Airblower1 := FALSE;
   Program16.NextStep1 := FALSE;
   Program16.PressureP1 := FALSE;
   Program16.SpareByte2H1 := 16#00;
   Program16.Revolution1 := 0;
   Program16.RopeUnit1_1 := 16#00;
   Program16.RopeUnit1_2 := 16#00;
   Program16.FilmForce1 := 0;
   Program16.FilmPrestretch1 := 0;
   Program16.Spare3H1 := 0;
   Program16.Spare49 := 0;
   Program16.Spare50 := 0;
   Program16.Spare51 := 0;
   Program16.Spare52 := 0;
   Program16.Spare53 := 0;
   Program16.Overlap1_2 := 0;
   Program16.Height2 := 0;
   Program16.Landmark2 := FALSE;
   Program16.Lifter2 := FALSE;
   Program16.SpareBit1H2 := FALSE;
   Program16.Airblower2 := FALSE;
   Program16.NextStep2 := FALSE;
   Program16.PressureP2 := FALSE;
   Program16.SpareByte2H2 := 16#00;
   Program16.Revolution2 := 0;
   Program16.RopeUnit2_1 := 16#00;
   Program16.RopeUnit2_2 := 16#00;
   Program16.FilmForce2 := 0;
   Program16.FilmPrestretch2 := 0;
   Program16.Spare3H2 := 0;
   Program16.Spare54 := 0;
   Program16.Spare55 := 0;
   Program16.Spare56 := 0;
   Program16.Spare57 := 0;
   Program16.Spare58 := 0;
   Program16.Overlap2_3 := 0;
   Program16.Height3 := 0;
   Program16.Landmark3 := FALSE;
   Program16.Lifter3 := FALSE;
   Program16.SpareBit1H3 := FALSE;
   Program16.Airblower3 := FALSE;
   Program16.NextStep3 := FALSE;
   Program16.PressureP3 := FALSE;
   Program16.SpareByte2H3 := 16#00;
   Program16.Revolution3 := 0;
   Program16.RopeUnit3_1 := 16#00;
   Program16.RopeUnit3_2 := 16#00;
   Program16.FilmForce3 := 0;
   Program16.FilmPrestretch3 := 0;
   Program16.Spare3H3 := 0;
   Program16.Spare59 := 0;
   Program16.Spare60 := 0;
   Program16.Spare61 := 0;
   Program16.Spare62 := 0;
   Program16.Spare63 := 0;
   Program16.Overlap3_4 := 0;
   Program16.Height4 := 0;
   Program16.Landmark4 := FALSE;
   Program16.Lifter4 := FALSE;
   Program16.SpareBit1H4 := FALSE;
   Program16.Airblower4 := FALSE;
   Program16.NextStep4 := FALSE;
   Program16.PressureP4 := FALSE;
   Program16.SpareByte2H4 := 16#00;
   Program16.Revolution4 := 0;
   Program16.RopeUnit4_1 := 16#00;
   Program16.RopeUnit4_2 := 16#00;
   Program16.FilmForce4 := 0;
   Program16.FilmPrestretch4 := 0;
   Program16.Spare3H4 := 0;
   Program16.Spare64 := 0;
   Program16.Spare65 := 0;
   Program16.Spare66 := 0;
   Program16.Spare67 := 0;
   Program16.Spare68 := 0;
   Program16.Overlap4_5 := 0;
   Program16.Height5 := 0;
   Program16.Landmark5 := FALSE;
   Program16.Lifter5 := FALSE;
   Program16.SpareBit1H5 := FALSE;
   Program16.Airblower5 := FALSE;
   Program16.NextStep5 := FALSE;
   Program16.PressureP5 := FALSE;
   Program16.SpareByte2H5 := 16#00;
   Program16.Revolution5 := 0;
   Program16.RopeUnit5_1 := 16#00;
   Program16.RopeUnit5_2 := 16#00;
   Program16.FilmForce5 := 0;
   Program16.FilmPrestretch5 := 0;
   Program16.Spare3H5 := 0;
   Program16.Spare69 := 0;
   Program16.Spare70 := 0;
   Program16.Spare71 := 0;
   Program16.Spare72 := 0;
   Program16.Spare73 := 0;
   Program16.Overlap5_6 := 0;
   Program16.Height6 := 0;
   Program16.Landmark6 := FALSE;
   Program16.Lifter6 := FALSE;
   Program16.SpareBit1H6 := FALSE;
   Program16.Airblower6 := FALSE;
   Program16.NextStep6 := FALSE;
   Program16.PressureP6 := FALSE;
   Program16.SpareByte2H6 := 16#00;
   Program16.Revolution6 := 0;
   Program16.RopeUnit6_1 := 16#00;
   Program16.RopeUnit6_2 := 16#00;
   Program16.FilmForce6 := 0;
   Program16.FilmPrestretch6 := 0;
   Program16.Spare3H6 := 0;
   Program16.Spare74 := 0;
   Program16.Spare75 := 0;
   Program16.Spare76 := 0;
   Program16.Spare77 := 0;
   Program16.Spare78 := 0;
   Program16.Overlap6_7 := 0;
   Program16.Height7 := 0;
   Program16.Landmark7 := FALSE;
   Program16.Lifter7 := FALSE;
   Program16.SpareBit1H7 := FALSE;
   Program16.Airblower7 := FALSE;
   Program16.NextStep7 := FALSE;
   Program16.PressureP7 := FALSE;
   Program16.SpareByte2H7 := 16#00;
   Program16.Revolution7 := 0;
   Program16.RopeUnit7_1 := 16#00;
   Program16.RopeUnit7_2 := 16#00;
   Program16.FilmForce7 := 0;
   Program16.FilmPrestretch7 := 0;
   Program16.Spare3H7 := 0;
   Program16.Spare79 := 0;
   Program16.Spare80 := 0;
   Program16.Spare81 := 0;
   Program16.Spare82 := 0;
   Program16.Spare83 := 0;
   Program16.Overlap7_8 := 0;
   Program16.Height8 := 0;
   Program16.Landmark8 := FALSE;
   Program16.Lifter8 := FALSE;
   Program16.SpareBit1H8 := FALSE;
   Program16.Airblower8 := FALSE;
   Program16.NextStep8 := FALSE;
   Program16.PressureP8 := FALSE;
   Program16.SpareByte2H8 := 16#00;
   Program16.Revolution8 := 0;
   Program16.RopeUnit8_1 := 16#00;
   Program16.RopeUnit8_2 := 16#00;
   Program16.FilmForce8 := 0;
   Program16.FilmPrestretch8 := 0;
   Program16.Spare3H8 := 0;
   Program16.Spare84 := 0;
   Program16.Spare85 := 0;
   Program16.Spare86 := 0;
   Program16.Spare87 := 0;
   Program16.Spare88 := 0;
   Program16.Overlap8_9 := 0;
   Program16.Height9 := 0;
   Program16.Landmark9 := FALSE;
   Program16.Lifter9 := FALSE;
   Program16.SpareBit1H9 := FALSE;
   Program16.Airblower9 := FALSE;
   Program16.NextStep9 := FALSE;
   Program16.PressureP9 := FALSE;
   Program16.SpareByte2H9 := 16#00;
   Program16.Revolution9 := 0;
   Program16.RopeUnit9_1 := 16#00;
   Program16.RopeUnit9_2 := 16#00;
   Program16.FilmForce9 := 0;
   Program16.FilmPrestretch9 := 0;
   Program16.Spare3H9 := 0;
   Program16.Spare89 := 0;
   Program16.Spare90 := 0;
   Program16.Spare91 := 0;
   Program16.Spare92 := 0;
   Program16.Spare93 := 0;
   Program16.Overlap9_10 := 0;
   Program16.Height10 := 0;
   Program16.Landmark10 := FALSE;
   Program16.Lifter10 := FALSE;
   Program16.SpareBit1H10 := FALSE;
   Program16.Airblower10 := FALSE;
   Program16.NextStep10 := FALSE;
   Program16.PressureP10 := FALSE;
   Program16.SpareByte2H10 := 16#00;
   Program16.Revolution10 := 0;
   Program16.RopeUnit10_1 := 16#00;
   Program16.RopeUnit10_2 := 16#00;
   Program16.FilmForce10 := 0;
   Program16.FilmPrestretch10 := 0;
   Program16.Spare3H10 := 0;
   Program16.Spare94 := 0;
   Program16.Spare95 := 0;
   Program16.Spare96 := 0;
   Program16.Spare97 := 0;
   Program16.Spare98 := 0;
   Program16.Overlap10_11 := 0;
   Program16.Height11 := 0;
   Program16.Landmark11 := FALSE;
   Program16.Lifter11 := FALSE;
   Program16.SpareBit1H11 := FALSE;
   Program16.Airblower11 := FALSE;
   Program16.NextStep11 := FALSE;
   Program16.PressureP11 := FALSE;
   Program16.SpareByte2H11 := 16#00;
   Program16.Revolution11 := 0;
   Program16.RopeUnit11_1 := 16#00;
   Program16.RopeUnit11_2 := 16#00;
   Program16.FilmForce11 := 0;
   Program16.FilmPrestretch11 := 0;
   Program16.Spare3H11 := 0;
   Program16.Spare99 := 0;
   Program16.Spare100 := 0;
   Program16.Spare101 := 0;
   Program16.Spare102 := 0;
   Program16.Spare103 := 0;
   Program16.Overlap11_12 := 0;
   Program16.Height12 := 0;
   Program16.Landmark12 := FALSE;
   Program16.Lifter12 := FALSE;
   Program16.SpareBit1H12 := FALSE;
   Program16.Airblower12 := FALSE;
   Program16.NextStep12 := FALSE;
   Program16.PressureP12 := FALSE;
   Program16.SpareByte2H12 := 16#00;
   Program16.Revolution12 := 0;
   Program16.RopeUnit12_1 := 16#00;
   Program16.RopeUnit12_2 := 16#00;
   Program16.FilmForce12 := 0;
   Program16.FilmPrestretch12 := 0;
   Program16.Spare3H12 := 0;
   Program16.Spare104 := 0;
   Program16.Spare105 := 0;
   Program16.Spare106 := 0;
   Program16.Spare107 := 0;
   Program16.Spare108 := 0;
END_DATA_BLOCK

DATA_BLOCK "DB235_Program15"   // DB235
{ S7_Optimized_Access := 'FALSE' }
AUTHOR : Robopac
VERSION : 0.0
// stored: AutoNumber false, IsOnlyStoredInLoadMemory false, IsWriteProtectedInAS false
   VAR RETAIN
      Program15 { S7_SetPoint := 'True'} : "DatiProgramma";
   END_VAR
BEGIN
   Program15.Wrapping := TRUE;
   Program15.TopLenght := 500;
   Program15.TopRelease := 0;
   Program15.TopDown := 0;
   Program15.Top := 4;
   Program15.PressurePTime := 0;
   Program15.LifterTime := 0;
   Program15.RevOverContrast := 1;
   Program15.RopeEndCycle := 16#02;
   Program15.Spare4 := 16#01;
   Program15.RopeTime := 1500;
   Program15.RevOverClamp := 1;
   Program15.FilmForceFinalRev := 10;
   Program15.FilmPrestretchFinalRev := 100;
   Program15.ArmSpeed := 100;
   Program15.CarriageDown4Top := 500;
   Program15.TopDownTime := 1500;
   Program15.LapsUnderTop := 0;
   Program15.Spare6 := 0;
   Program15.Spare7 := 0;
   Program15.Spare8 := 0;
   Program15.Spare9 := 0;
   Program15.Spare10 := 0;
   Program15.Spare11 := 0;
   Program15.Spare12 := 0;
   Program15.Overlap0_1 := 0;
   Program15.Height1 := 130;
   Program15.Landmark1 := FALSE;
   Program15.Lifter1 := FALSE;
   Program15.SpareBit1H1 := FALSE;
   Program15.Airblower1 := TRUE;
   Program15.NextStep1 := TRUE;
   Program15.PressureP1 := TRUE;
   Program15.SpareByte2H1 := 16#00;
   Program15.Revolution1 := 1;
   Program15.RopeUnit1_1 := 16#01;
   Program15.RopeUnit1_2 := 16#01;
   Program15.FilmForce1 := 5;
   Program15.FilmPrestretch1 := 200;
   Program15.Spare3H1 := 0;
   Program15.Spare49 := 0;
   Program15.Spare50 := 0;
   Program15.Spare51 := 0;
   Program15.Spare52 := 0;
   Program15.Spare53 := 0;
   Program15.Overlap1_2 := 0;
   Program15.Height2 := 50;
   Program15.Landmark2 := FALSE;
   Program15.Lifter2 := FALSE;
   Program15.SpareBit1H2 := FALSE;
   Program15.Airblower2 := TRUE;
   Program15.NextStep2 := TRUE;
   Program15.PressureP2 := TRUE;
   Program15.SpareByte2H2 := 16#00;
   Program15.Revolution2 := 1;
   Program15.RopeUnit2_1 := 16#01;
   Program15.RopeUnit2_2 := 16#01;
   Program15.FilmForce2 := 20;
   Program15.FilmPrestretch2 := 200;
   Program15.Spare3H2 := 0;
   Program15.Spare54 := 0;
   Program15.Spare55 := 0;
   Program15.Spare56 := 0;
   Program15.Spare57 := 0;
   Program15.Spare58 := 0;
   Program15.Overlap2_3 := 100;
   Program15.Height3 := -50;
   Program15.Landmark3 := TRUE;
   Program15.Lifter3 := FALSE;
   Program15.SpareBit1H3 := FALSE;
   Program15.Airblower3 := TRUE;
   Program15.NextStep3 := TRUE;
   Program15.PressureP3 := TRUE;
   Program15.SpareByte2H3 := 16#00;
   Program15.Revolution3 := 2;
   Program15.RopeUnit3_1 := 16#01;
   Program15.RopeUnit3_2 := 16#01;
   Program15.FilmForce3 := 30;
   Program15.FilmPrestretch3 := 200;
   Program15.Spare3H3 := 0;
   Program15.Spare59 := 0;
   Program15.Spare60 := 0;
   Program15.Spare61 := 380;
   Program15.Spare62 := 2800;
   Program15.Spare63 := 0;
   Program15.Overlap3_4 := 100;
   Program15.Height4 := 100;
   Program15.Landmark4 := FALSE;
   Program15.Lifter4 := FALSE;
   Program15.SpareBit1H4 := FALSE;
   Program15.Airblower4 := TRUE;
   Program15.NextStep4 := TRUE;
   Program15.PressureP4 := TRUE;
   Program15.SpareByte2H4 := 16#00;
   Program15.Revolution4 := 3;
   Program15.RopeUnit4_1 := 16#02;
   Program15.RopeUnit4_2 := 16#02;
   Program15.FilmForce4 := 30;
   Program15.FilmPrestretch4 := 200;
   Program15.Spare3H4 := 0;
   Program15.Spare64 := 0;
   Program15.Spare65 := 0;
   Program15.Spare66 := 0;
   Program15.Spare67 := 0;
   Program15.Spare68 := 0;
   Program15.Overlap4_5 := 0;
   Program15.Height5 := 50;
   Program15.Landmark5 := FALSE;
   Program15.Lifter5 := FALSE;
   Program15.SpareBit1H5 := FALSE;
   Program15.Airblower5 := TRUE;
   Program15.NextStep5 := FALSE;
   Program15.PressureP5 := FALSE;
   Program15.SpareByte2H5 := 16#00;
   Program15.Revolution5 := 1;
   Program15.RopeUnit5_1 := 16#01;
   Program15.RopeUnit5_2 := 16#01;
   Program15.FilmForce5 := 30;
   Program15.FilmPrestretch5 := 200;
   Program15.Spare3H5 := 0;
   Program15.Spare69 := 0;
   Program15.Spare70 := 0;
   Program15.Spare71 := 0;
   Program15.Spare72 := 0;
   Program15.Spare73 := 0;
   Program15.Overlap5_6 := 100;
   Program15.Height6 := 50;
   Program15.Landmark6 := FALSE;
   Program15.Lifter6 := FALSE;
   Program15.SpareBit1H6 := FALSE;
   Program15.Airblower6 := TRUE;
   Program15.NextStep6 := FALSE;
   Program15.PressureP6 := FALSE;
   Program15.SpareByte2H6 := 16#00;
   Program15.Revolution6 := 2;
   Program15.RopeUnit6_1 := 16#02;
   Program15.RopeUnit6_2 := 16#01;
   Program15.FilmForce6 := 20;
   Program15.FilmPrestretch6 := 200;
   Program15.Spare3H6 := 0;
   Program15.Spare74 := 0;
   Program15.Spare75 := 0;
   Program15.Spare76 := 0;
   Program15.Spare77 := 0;
   Program15.Spare78 := 0;
   Program15.Overlap6_7 := 0;
   Program15.Height7 := 0;
   Program15.Landmark7 := FALSE;
   Program15.Lifter7 := FALSE;
   Program15.SpareBit1H7 := FALSE;
   Program15.Airblower7 := FALSE;
   Program15.NextStep7 := TRUE;
   Program15.PressureP7 := FALSE;
   Program15.SpareByte2H7 := 16#00;
   Program15.Revolution7 := 1;
   Program15.RopeUnit7_1 := 16#01;
   Program15.RopeUnit7_2 := 16#01;
   Program15.FilmForce7 := 0;
   Program15.FilmPrestretch7 := 100;
   Program15.Spare3H7 := 0;
   Program15.Spare79 := 0;
   Program15.Spare80 := 0;
   Program15.Spare81 := 0;
   Program15.Spare82 := 0;
   Program15.Spare83 := 0;
   Program15.Overlap7_8 := 0;
   Program15.Height8 := 0;
   Program15.Landmark8 := FALSE;
   Program15.Lifter8 := FALSE;
   Program15.SpareBit1H8 := FALSE;
   Program15.Airblower8 := FALSE;
   Program15.NextStep8 := TRUE;
   Program15.PressureP8 := FALSE;
   Program15.SpareByte2H8 := 16#00;
   Program15.Revolution8 := 1;
   Program15.RopeUnit8_1 := 16#01;
   Program15.RopeUnit8_2 := 16#01;
   Program15.FilmForce8 := 0;
   Program15.FilmPrestretch8 := 100;
   Program15.Spare3H8 := 0;
   Program15.Spare84 := 0;
   Program15.Spare85 := 0;
   Program15.Spare86 := 0;
   Program15.Spare87 := 0;
   Program15.Spare88 := 0;
   Program15.Overlap8_9 := 0;
   Program15.Height9 := 0;
   Program15.Landmark9 := FALSE;
   Program15.Lifter9 := FALSE;
   Program15.SpareBit1H9 := FALSE;
   Program15.Airblower9 := FALSE;
   Program15.NextStep9 := TRUE;
   Program15.PressureP9 := FALSE;
   Program15.SpareByte2H9 := 16#00;
   Program15.Revolution9 := 1;
   Program15.RopeUnit9_1 := 16#01;
   Program15.RopeUnit9_2 := 16#01;
   Program15.FilmForce9 := 0;
   Program15.FilmPrestretch9 := 100;
   Program15.Spare3H9 := 0;
   Program15.Spare89 := 0;
   Program15.Spare90 := 0;
   Program15.Spare91 := 0;
   Program15.Spare92 := 0;
   Program15.Spare93 := 0;
   Program15.Overlap9_10 := 0;
   Program15.Height10 := 0;
   Program15.Landmark10 := FALSE;
   Program15.Lifter10 := FALSE;
   Program15.SpareBit1H10 := FALSE;
   Program15.Airblower10 := FALSE;
   Program15.NextStep10 := FALSE;
   Program15.PressureP10 := FALSE;
   Program15.SpareByte2H10 := 16#00;
   Program15.Revolution10 := 1;
   Program15.RopeUnit10_1 := 16#01;
   Program15.RopeUnit10_2 := 16#01;
   Program15.FilmForce10 := 0;
   Program15.FilmPrestretch10 := 100;
   Program15.Spare3H10 := 0;
   Program15.Spare94 := 0;
   Program15.Spare95 := 0;
   Program15.Spare96 := 0;
   Program15.Spare97 := 0;
   Program15.Spare98 := 0;
   Program15.Overlap10_11 := 0;
   Program15.Height11 := 0;
   Program15.Landmark11 := FALSE;
   Program15.Lifter11 := FALSE;
   Program15.SpareBit1H11 := FALSE;
   Program15.Airblower11 := FALSE;
   Program15.NextStep11 := TRUE;
   Program15.PressureP11 := FALSE;
   Program15.SpareByte2H11 := 16#00;
   Program15.Revolution11 := 1;
   Program15.RopeUnit11_1 := 16#01;
   Program15.RopeUnit11_2 := 16#01;
   Program15.FilmForce11 := 0;
   Program15.FilmPrestretch11 := 100;
   Program15.Spare3H11 := 0;
   Program15.Spare99 := 0;
   Program15.Spare100 := 0;
   Program15.Spare101 := 0;
   Program15.Spare102 := 0;
   Program15.Spare103 := 0;
   Program15.Overlap11_12 := 0;
   Program15.Height12 := 0;
   Program15.Landmark12 := FALSE;
   Program15.Lifter12 := FALSE;
   Program15.SpareBit1H12 := FALSE;
   Program15.Airblower12 := FALSE;
   Program15.NextStep12 := FALSE;
   Program15.PressureP12 := FALSE;
   Program15.SpareByte2H12 := 16#00;
   Program15.Revolution12 := 1;
   Program15.RopeUnit12_1 := 16#01;
   Program15.RopeUnit12_2 := 16#01;
   Program15.FilmForce12 := 0;
   Program15.FilmPrestretch12 := 100;
   Program15.Spare3H12 := 0;
   Program15.Spare104 := 0;
   Program15.Spare105 := 0;
   Program15.Spare106 := 0;
   Program15.Spare107 := 0;
   Program15.Spare108 := 0;
END_DATA_BLOCK

DATA_BLOCK "DB236_Program14"   // DB236
{ S7_Optimized_Access := 'FALSE' }
AUTHOR : Robopac
VERSION : 0.0
// stored: AutoNumber false, IsOnlyStoredInLoadMemory false, IsWriteProtectedInAS false
   VAR RETAIN
      Program14 { S7_SetPoint := 'True'} : "DatiProgramma";
   END_VAR
BEGIN
   Program14.Wrapping := TRUE;
   Program14.TopLenght := 500;
   Program14.TopRelease := 0;
   Program14.TopDown := 0;
   Program14.Top := 4;
   Program14.PressurePTime := 0;
   Program14.LifterTime := 0;
   Program14.RevOverContrast := 1;
   Program14.RopeEndCycle := 16#02;
   Program14.Spare4 := 16#01;
   Program14.RopeTime := 1500;
   Program14.RevOverClamp := 1;
   Program14.FilmForceFinalRev := 10;
   Program14.FilmPrestretchFinalRev := 100;
   Program14.ArmSpeed := 100;
   Program14.CarriageDown4Top := 500;
   Program14.TopDownTime := 1500;
   Program14.LapsUnderTop := 0;
   Program14.Spare6 := 0;
   Program14.Spare7 := 0;
   Program14.Spare8 := 0;
   Program14.Spare9 := 0;
   Program14.Spare10 := 0;
   Program14.Spare11 := 0;
   Program14.Spare12 := 0;
   Program14.Overlap0_1 := 0;
   Program14.Height1 := 130;
   Program14.Landmark1 := FALSE;
   Program14.Lifter1 := FALSE;
   Program14.SpareBit1H1 := FALSE;
   Program14.Airblower1 := TRUE;
   Program14.NextStep1 := TRUE;
   Program14.PressureP1 := TRUE;
   Program14.SpareByte2H1 := 16#00;
   Program14.Revolution1 := 1;
   Program14.RopeUnit1_1 := 16#01;
   Program14.RopeUnit1_2 := 16#01;
   Program14.FilmForce1 := 5;
   Program14.FilmPrestretch1 := 200;
   Program14.Spare3H1 := 0;
   Program14.Spare49 := 0;
   Program14.Spare50 := 0;
   Program14.Spare51 := 0;
   Program14.Spare52 := 0;
   Program14.Spare53 := 0;
   Program14.Overlap1_2 := 0;
   Program14.Height2 := 50;
   Program14.Landmark2 := FALSE;
   Program14.Lifter2 := FALSE;
   Program14.SpareBit1H2 := FALSE;
   Program14.Airblower2 := TRUE;
   Program14.NextStep2 := TRUE;
   Program14.PressureP2 := TRUE;
   Program14.SpareByte2H2 := 16#00;
   Program14.Revolution2 := 1;
   Program14.RopeUnit2_1 := 16#01;
   Program14.RopeUnit2_2 := 16#01;
   Program14.FilmForce2 := 20;
   Program14.FilmPrestretch2 := 200;
   Program14.Spare3H2 := 0;
   Program14.Spare54 := 0;
   Program14.Spare55 := 0;
   Program14.Spare56 := 0;
   Program14.Spare57 := 0;
   Program14.Spare58 := 0;
   Program14.Overlap2_3 := 100;
   Program14.Height3 := -50;
   Program14.Landmark3 := TRUE;
   Program14.Lifter3 := FALSE;
   Program14.SpareBit1H3 := FALSE;
   Program14.Airblower3 := TRUE;
   Program14.NextStep3 := TRUE;
   Program14.PressureP3 := TRUE;
   Program14.SpareByte2H3 := 16#00;
   Program14.Revolution3 := 2;
   Program14.RopeUnit3_1 := 16#01;
   Program14.RopeUnit3_2 := 16#01;
   Program14.FilmForce3 := 30;
   Program14.FilmPrestretch3 := 200;
   Program14.Spare3H3 := 0;
   Program14.Spare59 := 0;
   Program14.Spare60 := 0;
   Program14.Spare61 := 380;
   Program14.Spare62 := 2800;
   Program14.Spare63 := 0;
   Program14.Overlap3_4 := 100;
   Program14.Height4 := 100;
   Program14.Landmark4 := FALSE;
   Program14.Lifter4 := FALSE;
   Program14.SpareBit1H4 := FALSE;
   Program14.Airblower4 := TRUE;
   Program14.NextStep4 := TRUE;
   Program14.PressureP4 := TRUE;
   Program14.SpareByte2H4 := 16#00;
   Program14.Revolution4 := 3;
   Program14.RopeUnit4_1 := 16#02;
   Program14.RopeUnit4_2 := 16#02;
   Program14.FilmForce4 := 30;
   Program14.FilmPrestretch4 := 200;
   Program14.Spare3H4 := 0;
   Program14.Spare64 := 0;
   Program14.Spare65 := 0;
   Program14.Spare66 := 0;
   Program14.Spare67 := 0;
   Program14.Spare68 := 0;
   Program14.Overlap4_5 := 0;
   Program14.Height5 := 50;
   Program14.Landmark5 := FALSE;
   Program14.Lifter5 := FALSE;
   Program14.SpareBit1H5 := FALSE;
   Program14.Airblower5 := TRUE;
   Program14.NextStep5 := FALSE;
   Program14.PressureP5 := FALSE;
   Program14.SpareByte2H5 := 16#00;
   Program14.Revolution5 := 1;
   Program14.RopeUnit5_1 := 16#01;
   Program14.RopeUnit5_2 := 16#01;
   Program14.FilmForce5 := 30;
   Program14.FilmPrestretch5 := 200;
   Program14.Spare3H5 := 0;
   Program14.Spare69 := 0;
   Program14.Spare70 := 0;
   Program14.Spare71 := 0;
   Program14.Spare72 := 0;
   Program14.Spare73 := 0;
   Program14.Overlap5_6 := 100;
   Program14.Height6 := 50;
   Program14.Landmark6 := FALSE;
   Program14.Lifter6 := FALSE;
   Program14.SpareBit1H6 := FALSE;
   Program14.Airblower6 := TRUE;
   Program14.NextStep6 := FALSE;
   Program14.PressureP6 := FALSE;
   Program14.SpareByte2H6 := 16#00;
   Program14.Revolution6 := 2;
   Program14.RopeUnit6_1 := 16#02;
   Program14.RopeUnit6_2 := 16#01;
   Program14.FilmForce6 := 20;
   Program14.FilmPrestretch6 := 200;
   Program14.Spare3H6 := 0;
   Program14.Spare74 := 0;
   Program14.Spare75 := 0;
   Program14.Spare76 := 0;
   Program14.Spare77 := 0;
   Program14.Spare78 := 0;
   Program14.Overlap6_7 := 0;
   Program14.Height7 := 0;
   Program14.Landmark7 := FALSE;
   Program14.Lifter7 := FALSE;
   Program14.SpareBit1H7 := FALSE;
   Program14.Airblower7 := FALSE;
   Program14.NextStep7 := TRUE;
   Program14.PressureP7 := FALSE;
   Program14.SpareByte2H7 := 16#00;
   Program14.Revolution7 := 1;
   Program14.RopeUnit7_1 := 16#01;
   Program14.RopeUnit7_2 := 16#01;
   Program14.FilmForce7 := 0;
   Program14.FilmPrestretch7 := 100;
   Program14.Spare3H7 := 0;
   Program14.Spare79 := 0;
   Program14.Spare80 := 0;
   Program14.Spare81 := 0;
   Program14.Spare82 := 0;
   Program14.Spare83 := 0;
   Program14.Overlap7_8 := 0;
   Program14.Height8 := 0;
   Program14.Landmark8 := FALSE;
   Program14.Lifter8 := FALSE;
   Program14.SpareBit1H8 := FALSE;
   Program14.Airblower8 := FALSE;
   Program14.NextStep8 := TRUE;
   Program14.PressureP8 := FALSE;
   Program14.SpareByte2H8 := 16#00;
   Program14.Revolution8 := 1;
   Program14.RopeUnit8_1 := 16#01;
   Program14.RopeUnit8_2 := 16#01;
   Program14.FilmForce8 := 0;
   Program14.FilmPrestretch8 := 100;
   Program14.Spare3H8 := 0;
   Program14.Spare84 := 0;
   Program14.Spare85 := 0;
   Program14.Spare86 := 0;
   Program14.Spare87 := 0;
   Program14.Spare88 := 0;
   Program14.Overlap8_9 := 0;
   Program14.Height9 := 0;
   Program14.Landmark9 := FALSE;
   Program14.Lifter9 := FALSE;
   Program14.SpareBit1H9 := FALSE;
   Program14.Airblower9 := FALSE;
   Program14.NextStep9 := TRUE;
   Program14.PressureP9 := FALSE;
   Program14.SpareByte2H9 := 16#00;
   Program14.Revolution9 := 1;
   Program14.RopeUnit9_1 := 16#01;
   Program14.RopeUnit9_2 := 16#01;
   Program14.FilmForce9 := 0;
   Program14.FilmPrestretch9 := 100;
   Program14.Spare3H9 := 0;
   Program14.Spare89 := 0;
   Program14.Spare90 := 0;
   Program14.Spare91 := 0;
   Program14.Spare92 := 0;
   Program14.Spare93 := 0;
   Program14.Overlap9_10 := 0;
   Program14.Height10 := 0;
   Program14.Landmark10 := FALSE;
   Program14.Lifter10 := FALSE;
   Program14.SpareBit1H10 := FALSE;
   Program14.Airblower10 := FALSE;
   Program14.NextStep10 := FALSE;
   Program14.PressureP10 := FALSE;
   Program14.SpareByte2H10 := 16#00;
   Program14.Revolution10 := 1;
   Program14.RopeUnit10_1 := 16#01;
   Program14.RopeUnit10_2 := 16#01;
   Program14.FilmForce10 := 0;
   Program14.FilmPrestretch10 := 100;
   Program14.Spare3H10 := 0;
   Program14.Spare94 := 0;
   Program14.Spare95 := 0;
   Program14.Spare96 := 0;
   Program14.Spare97 := 0;
   Program14.Spare98 := 0;
   Program14.Overlap10_11 := 0;
   Program14.Height11 := 0;
   Program14.Landmark11 := FALSE;
   Program14.Lifter11 := FALSE;
   Program14.SpareBit1H11 := FALSE;
   Program14.Airblower11 := FALSE;
   Program14.NextStep11 := TRUE;
   Program14.PressureP11 := FALSE;
   Program14.SpareByte2H11 := 16#00;
   Program14.Revolution11 := 1;
   Program14.RopeUnit11_1 := 16#01;
   Program14.RopeUnit11_2 := 16#01;
   Program14.FilmForce11 := 0;
   Program14.FilmPrestretch11 := 100;
   Program14.Spare3H11 := 0;
   Program14.Spare99 := 0;
   Program14.Spare100 := 0;
   Program14.Spare101 := 0;
   Program14.Spare102 := 0;
   Program14.Spare103 := 0;
   Program14.Overlap11_12 := 0;
   Program14.Height12 := 0;
   Program14.Landmark12 := FALSE;
   Program14.Lifter12 := FALSE;
   Program14.SpareBit1H12 := FALSE;
   Program14.Airblower12 := FALSE;
   Program14.NextStep12 := FALSE;
   Program14.PressureP12 := FALSE;
   Program14.SpareByte2H12 := 16#00;
   Program14.Revolution12 := 1;
   Program14.RopeUnit12_1 := 16#01;
   Program14.RopeUnit12_2 := 16#01;
   Program14.FilmForce12 := 0;
   Program14.FilmPrestretch12 := 100;
   Program14.Spare3H12 := 0;
   Program14.Spare104 := 0;
   Program14.Spare105 := 0;
   Program14.Spare106 := 0;
   Program14.Spare107 := 0;
   Program14.Spare108 := 0;
END_DATA_BLOCK

DATA_BLOCK "DB237_Program13"   // DB237
{ S7_Optimized_Access := 'FALSE' }
AUTHOR : Robopac
VERSION : 0.0
// stored: AutoNumber false, IsOnlyStoredInLoadMemory false, IsWriteProtectedInAS false
   VAR RETAIN
      Program13 { S7_SetPoint := 'True'} : "DatiProgramma";
   END_VAR
BEGIN
   Program13.Wrapping := TRUE;
   Program13.TopLenght := 500;
   Program13.TopRelease := 0;
   Program13.TopDown := 0;
   Program13.Top := 4;
   Program13.PressurePTime := 0;
   Program13.LifterTime := 0;
   Program13.RevOverContrast := 1;
   Program13.RopeEndCycle := 16#02;
   Program13.Spare4 := 16#01;
   Program13.RopeTime := 1500;
   Program13.RevOverClamp := 1;
   Program13.FilmForceFinalRev := 10;
   Program13.FilmPrestretchFinalRev := 100;
   Program13.ArmSpeed := 100;
   Program13.CarriageDown4Top := 500;
   Program13.TopDownTime := 1500;
   Program13.LapsUnderTop := 0;
   Program13.Spare6 := 0;
   Program13.Spare7 := 0;
   Program13.Spare8 := 0;
   Program13.Spare9 := 0;
   Program13.Spare10 := 0;
   Program13.Spare11 := 0;
   Program13.Spare12 := 0;
   Program13.Overlap0_1 := 0;
   Program13.Height1 := 130;
   Program13.Landmark1 := FALSE;
   Program13.Lifter1 := FALSE;
   Program13.SpareBit1H1 := FALSE;
   Program13.Airblower1 := TRUE;
   Program13.NextStep1 := TRUE;
   Program13.PressureP1 := TRUE;
   Program13.SpareByte2H1 := 16#00;
   Program13.Revolution1 := 1;
   Program13.RopeUnit1_1 := 16#01;
   Program13.RopeUnit1_2 := 16#01;
   Program13.FilmForce1 := 5;
   Program13.FilmPrestretch1 := 200;
   Program13.Spare3H1 := 0;
   Program13.Spare49 := 0;
   Program13.Spare50 := 0;
   Program13.Spare51 := 0;
   Program13.Spare52 := 0;
   Program13.Spare53 := 0;
   Program13.Overlap1_2 := 0;
   Program13.Height2 := 50;
   Program13.Landmark2 := FALSE;
   Program13.Lifter2 := FALSE;
   Program13.SpareBit1H2 := FALSE;
   Program13.Airblower2 := TRUE;
   Program13.NextStep2 := TRUE;
   Program13.PressureP2 := TRUE;
   Program13.SpareByte2H2 := 16#00;
   Program13.Revolution2 := 1;
   Program13.RopeUnit2_1 := 16#01;
   Program13.RopeUnit2_2 := 16#01;
   Program13.FilmForce2 := 20;
   Program13.FilmPrestretch2 := 200;
   Program13.Spare3H2 := 0;
   Program13.Spare54 := 0;
   Program13.Spare55 := 0;
   Program13.Spare56 := 0;
   Program13.Spare57 := 0;
   Program13.Spare58 := 0;
   Program13.Overlap2_3 := 100;
   Program13.Height3 := -50;
   Program13.Landmark3 := TRUE;
   Program13.Lifter3 := FALSE;
   Program13.SpareBit1H3 := FALSE;
   Program13.Airblower3 := TRUE;
   Program13.NextStep3 := TRUE;
   Program13.PressureP3 := TRUE;
   Program13.SpareByte2H3 := 16#00;
   Program13.Revolution3 := 2;
   Program13.RopeUnit3_1 := 16#01;
   Program13.RopeUnit3_2 := 16#01;
   Program13.FilmForce3 := 30;
   Program13.FilmPrestretch3 := 200;
   Program13.Spare3H3 := 0;
   Program13.Spare59 := 0;
   Program13.Spare60 := 0;
   Program13.Spare61 := 380;
   Program13.Spare62 := 2800;
   Program13.Spare63 := 0;
   Program13.Overlap3_4 := 100;
   Program13.Height4 := 100;
   Program13.Landmark4 := FALSE;
   Program13.Lifter4 := FALSE;
   Program13.SpareBit1H4 := FALSE;
   Program13.Airblower4 := TRUE;
   Program13.NextStep4 := TRUE;
   Program13.PressureP4 := TRUE;
   Program13.SpareByte2H4 := 16#00;
   Program13.Revolution4 := 3;
   Program13.RopeUnit4_1 := 16#02;
   Program13.RopeUnit4_2 := 16#02;
   Program13.FilmForce4 := 30;
   Program13.FilmPrestretch4 := 200;
   Program13.Spare3H4 := 0;
   Program13.Spare64 := 0;
   Program13.Spare65 := 0;
   Program13.Spare66 := 0;
   Program13.Spare67 := 0;
   Program13.Spare68 := 0;
   Program13.Overlap4_5 := 0;
   Program13.Height5 := 50;
   Program13.Landmark5 := FALSE;
   Program13.Lifter5 := FALSE;
   Program13.SpareBit1H5 := FALSE;
   Program13.Airblower5 := TRUE;
   Program13.NextStep5 := FALSE;
   Program13.PressureP5 := FALSE;
   Program13.SpareByte2H5 := 16#00;
   Program13.Revolution5 := 1;
   Program13.RopeUnit5_1 := 16#01;
   Program13.RopeUnit5_2 := 16#01;
   Program13.FilmForce5 := 30;
   Program13.FilmPrestretch5 := 200;
   Program13.Spare3H5 := 0;
   Program13.Spare69 := 0;
   Program13.Spare70 := 0;
   Program13.Spare71 := 0;
   Program13.Spare72 := 0;
   Program13.Spare73 := 0;
   Program13.Overlap5_6 := 100;
   Program13.Height6 := 50;
   Program13.Landmark6 := FALSE;
   Program13.Lifter6 := FALSE;
   Program13.SpareBit1H6 := FALSE;
   Program13.Airblower6 := TRUE;
   Program13.NextStep6 := FALSE;
   Program13.PressureP6 := FALSE;
   Program13.SpareByte2H6 := 16#00;
   Program13.Revolution6 := 2;
   Program13.RopeUnit6_1 := 16#02;
   Program13.RopeUnit6_2 := 16#01;
   Program13.FilmForce6 := 20;
   Program13.FilmPrestretch6 := 200;
   Program13.Spare3H6 := 0;
   Program13.Spare74 := 0;
   Program13.Spare75 := 0;
   Program13.Spare76 := 0;
   Program13.Spare77 := 0;
   Program13.Spare78 := 0;
   Program13.Overlap6_7 := 0;
   Program13.Height7 := 0;
   Program13.Landmark7 := FALSE;
   Program13.Lifter7 := FALSE;
   Program13.SpareBit1H7 := FALSE;
   Program13.Airblower7 := FALSE;
   Program13.NextStep7 := TRUE;
   Program13.PressureP7 := FALSE;
   Program13.SpareByte2H7 := 16#00;
   Program13.Revolution7 := 1;
   Program13.RopeUnit7_1 := 16#01;
   Program13.RopeUnit7_2 := 16#01;
   Program13.FilmForce7 := 0;
   Program13.FilmPrestretch7 := 100;
   Program13.Spare3H7 := 0;
   Program13.Spare79 := 0;
   Program13.Spare80 := 0;
   Program13.Spare81 := 0;
   Program13.Spare82 := 0;
   Program13.Spare83 := 0;
   Program13.Overlap7_8 := 0;
   Program13.Height8 := 0;
   Program13.Landmark8 := FALSE;
   Program13.Lifter8 := FALSE;
   Program13.SpareBit1H8 := FALSE;
   Program13.Airblower8 := FALSE;
   Program13.NextStep8 := TRUE;
   Program13.PressureP8 := FALSE;
   Program13.SpareByte2H8 := 16#00;
   Program13.Revolution8 := 1;
   Program13.RopeUnit8_1 := 16#01;
   Program13.RopeUnit8_2 := 16#01;
   Program13.FilmForce8 := 0;
   Program13.FilmPrestretch8 := 100;
   Program13.Spare3H8 := 0;
   Program13.Spare84 := 0;
   Program13.Spare85 := 0;
   Program13.Spare86 := 0;
   Program13.Spare87 := 0;
   Program13.Spare88 := 0;
   Program13.Overlap8_9 := 0;
   Program13.Height9 := 0;
   Program13.Landmark9 := FALSE;
   Program13.Lifter9 := FALSE;
   Program13.SpareBit1H9 := FALSE;
   Program13.Airblower9 := FALSE;
   Program13.NextStep9 := TRUE;
   Program13.PressureP9 := FALSE;
   Program13.SpareByte2H9 := 16#00;
   Program13.Revolution9 := 1;
   Program13.RopeUnit9_1 := 16#01;
   Program13.RopeUnit9_2 := 16#01;
   Program13.FilmForce9 := 0;
   Program13.FilmPrestretch9 := 100;
   Program13.Spare3H9 := 0;
   Program13.Spare89 := 0;
   Program13.Spare90 := 0;
   Program13.Spare91 := 0;
   Program13.Spare92 := 0;
   Program13.Spare93 := 0;
   Program13.Overlap9_10 := 0;
   Program13.Height10 := 0;
   Program13.Landmark10 := FALSE;
   Program13.Lifter10 := FALSE;
   Program13.SpareBit1H10 := FALSE;
   Program13.Airblower10 := FALSE;
   Program13.NextStep10 := FALSE;
   Program13.PressureP10 := FALSE;
   Program13.SpareByte2H10 := 16#00;
   Program13.Revolution10 := 1;
   Program13.RopeUnit10_1 := 16#01;
   Program13.RopeUnit10_2 := 16#01;
   Program13.FilmForce10 := 0;
   Program13.FilmPrestretch10 := 100;
   Program13.Spare3H10 := 0;
   Program13.Spare94 := 0;
   Program13.Spare95 := 0;
   Program13.Spare96 := 0;
   Program13.Spare97 := 0;
   Program13.Spare98 := 0;
   Program13.Overlap10_11 := 0;
   Program13.Height11 := 0;
   Program13.Landmark11 := FALSE;
   Program13.Lifter11 := FALSE;
   Program13.SpareBit1H11 := FALSE;
   Program13.Airblower11 := FALSE;
   Program13.NextStep11 := TRUE;
   Program13.PressureP11 := FALSE;
   Program13.SpareByte2H11 := 16#00;
   Program13.Revolution11 := 1;
   Program13.RopeUnit11_1 := 16#01;
   Program13.RopeUnit11_2 := 16#01;
   Program13.FilmForce11 := 0;
   Program13.FilmPrestretch11 := 100;
   Program13.Spare3H11 := 0;
   Program13.Spare99 := 0;
   Program13.Spare100 := 0;
   Program13.Spare101 := 0;
   Program13.Spare102 := 0;
   Program13.Spare103 := 0;
   Program13.Overlap11_12 := 0;
   Program13.Height12 := 0;
   Program13.Landmark12 := FALSE;
   Program13.Lifter12 := FALSE;
   Program13.SpareBit1H12 := FALSE;
   Program13.Airblower12 := FALSE;
   Program13.NextStep12 := FALSE;
   Program13.PressureP12 := FALSE;
   Program13.SpareByte2H12 := 16#00;
   Program13.Revolution12 := 1;
   Program13.RopeUnit12_1 := 16#01;
   Program13.RopeUnit12_2 := 16#01;
   Program13.FilmForce12 := 0;
   Program13.FilmPrestretch12 := 100;
   Program13.Spare3H12 := 0;
   Program13.Spare104 := 0;
   Program13.Spare105 := 0;
   Program13.Spare106 := 0;
   Program13.Spare107 := 0;
   Program13.Spare108 := 0;
END_DATA_BLOCK

DATA_BLOCK "DB238_Program12"   // DB238
{ S7_Optimized_Access := 'FALSE' }
AUTHOR : Robopac
VERSION : 0.0
// stored: AutoNumber false, IsOnlyStoredInLoadMemory false, IsWriteProtectedInAS false
   VAR RETAIN
      Program12 { S7_SetPoint := 'True'} : "DatiProgramma";
   END_VAR
BEGIN
   Program12.Wrapping := TRUE;
   Program12.TopLenght := 500;
   Program12.TopRelease := 0;
   Program12.TopDown := 0;
   Program12.Top := 4;
   Program12.PressurePTime := 0;
   Program12.LifterTime := 0;
   Program12.RevOverContrast := 1;
   Program12.RopeEndCycle := 16#02;
   Program12.Spare4 := 16#01;
   Program12.RopeTime := 1500;
   Program12.RevOverClamp := 1;
   Program12.FilmForceFinalRev := 10;
   Program12.FilmPrestretchFinalRev := 100;
   Program12.ArmSpeed := 100;
   Program12.CarriageDown4Top := 500;
   Program12.TopDownTime := 1500;
   Program12.LapsUnderTop := 0;
   Program12.Spare6 := 0;
   Program12.Spare7 := 0;
   Program12.Spare8 := 0;
   Program12.Spare9 := 0;
   Program12.Spare10 := 0;
   Program12.Spare11 := 0;
   Program12.Spare12 := 0;
   Program12.Overlap0_1 := 0;
   Program12.Height1 := 130;
   Program12.Landmark1 := FALSE;
   Program12.Lifter1 := FALSE;
   Program12.SpareBit1H1 := FALSE;
   Program12.Airblower1 := TRUE;
   Program12.NextStep1 := TRUE;
   Program12.PressureP1 := TRUE;
   Program12.SpareByte2H1 := 16#00;
   Program12.Revolution1 := 1;
   Program12.RopeUnit1_1 := 16#01;
   Program12.RopeUnit1_2 := 16#01;
   Program12.FilmForce1 := 5;
   Program12.FilmPrestretch1 := 200;
   Program12.Spare3H1 := 0;
   Program12.Spare49 := 0;
   Program12.Spare50 := 0;
   Program12.Spare51 := 0;
   Program12.Spare52 := 0;
   Program12.Spare53 := 0;
   Program12.Overlap1_2 := 0;
   Program12.Height2 := 50;
   Program12.Landmark2 := FALSE;
   Program12.Lifter2 := FALSE;
   Program12.SpareBit1H2 := FALSE;
   Program12.Airblower2 := TRUE;
   Program12.NextStep2 := TRUE;
   Program12.PressureP2 := TRUE;
   Program12.SpareByte2H2 := 16#00;
   Program12.Revolution2 := 1;
   Program12.RopeUnit2_1 := 16#01;
   Program12.RopeUnit2_2 := 16#01;
   Program12.FilmForce2 := 20;
   Program12.FilmPrestretch2 := 200;
   Program12.Spare3H2 := 0;
   Program12.Spare54 := 0;
   Program12.Spare55 := 0;
   Program12.Spare56 := 0;
   Program12.Spare57 := 0;
   Program12.Spare58 := 0;
   Program12.Overlap2_3 := 100;
   Program12.Height3 := -50;
   Program12.Landmark3 := TRUE;
   Program12.Lifter3 := FALSE;
   Program12.SpareBit1H3 := FALSE;
   Program12.Airblower3 := TRUE;
   Program12.NextStep3 := TRUE;
   Program12.PressureP3 := TRUE;
   Program12.SpareByte2H3 := 16#00;
   Program12.Revolution3 := 2;
   Program12.RopeUnit3_1 := 16#01;
   Program12.RopeUnit3_2 := 16#01;
   Program12.FilmForce3 := 30;
   Program12.FilmPrestretch3 := 200;
   Program12.Spare3H3 := 0;
   Program12.Spare59 := 0;
   Program12.Spare60 := 0;
   Program12.Spare61 := 380;
   Program12.Spare62 := 2800;
   Program12.Spare63 := 0;
   Program12.Overlap3_4 := 100;
   Program12.Height4 := 100;
   Program12.Landmark4 := FALSE;
   Program12.Lifter4 := FALSE;
   Program12.SpareBit1H4 := FALSE;
   Program12.Airblower4 := TRUE;
   Program12.NextStep4 := TRUE;
   Program12.PressureP4 := TRUE;
   Program12.SpareByte2H4 := 16#00;
   Program12.Revolution4 := 3;
   Program12.RopeUnit4_1 := 16#02;
   Program12.RopeUnit4_2 := 16#02;
   Program12.FilmForce4 := 30;
   Program12.FilmPrestretch4 := 200;
   Program12.Spare3H4 := 0;
   Program12.Spare64 := 0;
   Program12.Spare65 := 0;
   Program12.Spare66 := 0;
   Program12.Spare67 := 0;
   Program12.Spare68 := 0;
   Program12.Overlap4_5 := 0;
   Program12.Height5 := 50;
   Program12.Landmark5 := FALSE;
   Program12.Lifter5 := FALSE;
   Program12.SpareBit1H5 := FALSE;
   Program12.Airblower5 := TRUE;
   Program12.NextStep5 := FALSE;
   Program12.PressureP5 := FALSE;
   Program12.SpareByte2H5 := 16#00;
   Program12.Revolution5 := 1;
   Program12.RopeUnit5_1 := 16#01;
   Program12.RopeUnit5_2 := 16#01;
   Program12.FilmForce5 := 30;
   Program12.FilmPrestretch5 := 200;
   Program12.Spare3H5 := 0;
   Program12.Spare69 := 0;
   Program12.Spare70 := 0;
   Program12.Spare71 := 0;
   Program12.Spare72 := 0;
   Program12.Spare73 := 0;
   Program12.Overlap5_6 := 100;
   Program12.Height6 := 50;
   Program12.Landmark6 := FALSE;
   Program12.Lifter6 := FALSE;
   Program12.SpareBit1H6 := FALSE;
   Program12.Airblower6 := TRUE;
   Program12.NextStep6 := FALSE;
   Program12.PressureP6 := FALSE;
   Program12.SpareByte2H6 := 16#00;
   Program12.Revolution6 := 2;
   Program12.RopeUnit6_1 := 16#02;
   Program12.RopeUnit6_2 := 16#01;
   Program12.FilmForce6 := 20;
   Program12.FilmPrestretch6 := 200;
   Program12.Spare3H6 := 0;
   Program12.Spare74 := 0;
   Program12.Spare75 := 0;
   Program12.Spare76 := 0;
   Program12.Spare77 := 0;
   Program12.Spare78 := 0;
   Program12.Overlap6_7 := 0;
   Program12.Height7 := 0;
   Program12.Landmark7 := FALSE;
   Program12.Lifter7 := FALSE;
   Program12.SpareBit1H7 := FALSE;
   Program12.Airblower7 := FALSE;
   Program12.NextStep7 := TRUE;
   Program12.PressureP7 := FALSE;
   Program12.SpareByte2H7 := 16#00;
   Program12.Revolution7 := 1;
   Program12.RopeUnit7_1 := 16#01;
   Program12.RopeUnit7_2 := 16#01;
   Program12.FilmForce7 := 0;
   Program12.FilmPrestretch7 := 100;
   Program12.Spare3H7 := 0;
   Program12.Spare79 := 0;
   Program12.Spare80 := 0;
   Program12.Spare81 := 0;
   Program12.Spare82 := 0;
   Program12.Spare83 := 0;
   Program12.Overlap7_8 := 0;
   Program12.Height8 := 0;
   Program12.Landmark8 := FALSE;
   Program12.Lifter8 := FALSE;
   Program12.SpareBit1H8 := FALSE;
   Program12.Airblower8 := FALSE;
   Program12.NextStep8 := TRUE;
   Program12.PressureP8 := FALSE;
   Program12.SpareByte2H8 := 16#00;
   Program12.Revolution8 := 1;
   Program12.RopeUnit8_1 := 16#01;
   Program12.RopeUnit8_2 := 16#01;
   Program12.FilmForce8 := 0;
   Program12.FilmPrestretch8 := 100;
   Program12.Spare3H8 := 0;
   Program12.Spare84 := 0;
   Program12.Spare85 := 0;
   Program12.Spare86 := 0;
   Program12.Spare87 := 0;
   Program12.Spare88 := 0;
   Program12.Overlap8_9 := 0;
   Program12.Height9 := 0;
   Program12.Landmark9 := FALSE;
   Program12.Lifter9 := FALSE;
   Program12.SpareBit1H9 := FALSE;
   Program12.Airblower9 := FALSE;
   Program12.NextStep9 := TRUE;
   Program12.PressureP9 := FALSE;
   Program12.SpareByte2H9 := 16#00;
   Program12.Revolution9 := 1;
   Program12.RopeUnit9_1 := 16#01;
   Program12.RopeUnit9_2 := 16#01;
   Program12.FilmForce9 := 0;
   Program12.FilmPrestretch9 := 100;
   Program12.Spare3H9 := 0;
   Program12.Spare89 := 0;
   Program12.Spare90 := 0;
   Program12.Spare91 := 0;
   Program12.Spare92 := 0;
   Program12.Spare93 := 0;
   Program12.Overlap9_10 := 0;
   Program12.Height10 := 0;
   Program12.Landmark10 := FALSE;
   Program12.Lifter10 := FALSE;
   Program12.SpareBit1H10 := FALSE;
   Program12.Airblower10 := FALSE;
   Program12.NextStep10 := FALSE;
   Program12.PressureP10 := FALSE;
   Program12.SpareByte2H10 := 16#00;
   Program12.Revolution10 := 1;
   Program12.RopeUnit10_1 := 16#01;
   Program12.RopeUnit10_2 := 16#01;
   Program12.FilmForce10 := 0;
   Program12.FilmPrestretch10 := 100;
   Program12.Spare3H10 := 0;
   Program12.Spare94 := 0;
   Program12.Spare95 := 0;
   Program12.Spare96 := 0;
   Program12.Spare97 := 0;
   Program12.Spare98 := 0;
   Program12.Overlap10_11 := 0;
   Program12.Height11 := 0;
   Program12.Landmark11 := FALSE;
   Program12.Lifter11 := FALSE;
   Program12.SpareBit1H11 := FALSE;
   Program12.Airblower11 := FALSE;
   Program12.NextStep11 := TRUE;
   Program12.PressureP11 := FALSE;
   Program12.SpareByte2H11 := 16#00;
   Program12.Revolution11 := 1;
   Program12.RopeUnit11_1 := 16#01;
   Program12.RopeUnit11_2 := 16#01;
   Program12.FilmForce11 := 0;
   Program12.FilmPrestretch11 := 100;
   Program12.Spare3H11 := 0;
   Program12.Spare99 := 0;
   Program12.Spare100 := 0;
   Program12.Spare101 := 0;
   Program12.Spare102 := 0;
   Program12.Spare103 := 0;
   Program12.Overlap11_12 := 0;
   Program12.Height12 := 0;
   Program12.Landmark12 := FALSE;
   Program12.Lifter12 := FALSE;
   Program12.SpareBit1H12 := FALSE;
   Program12.Airblower12 := FALSE;
   Program12.NextStep12 := FALSE;
   Program12.PressureP12 := FALSE;
   Program12.SpareByte2H12 := 16#00;
   Program12.Revolution12 := 1;
   Program12.RopeUnit12_1 := 16#01;
   Program12.RopeUnit12_2 := 16#01;
   Program12.FilmForce12 := 0;
   Program12.FilmPrestretch12 := 100;
   Program12.Spare3H12 := 0;
   Program12.Spare104 := 0;
   Program12.Spare105 := 0;
   Program12.Spare106 := 0;
   Program12.Spare107 := 0;
   Program12.Spare108 := 0;
END_DATA_BLOCK

DATA_BLOCK "DB239_Program11"   // DB239
{ S7_Optimized_Access := 'FALSE' }
AUTHOR : Robopac
VERSION : 0.0
// stored: AutoNumber false, IsOnlyStoredInLoadMemory false, IsWriteProtectedInAS false
   VAR RETAIN
      Program11 { S7_SetPoint := 'True'} : "DatiProgramma";
   END_VAR
BEGIN
   Program11.Wrapping := TRUE;
   Program11.TopLenght := 500;
   Program11.TopRelease := 0;
   Program11.TopDown := 0;
   Program11.Top := 4;
   Program11.PressurePTime := 0;
   Program11.LifterTime := 0;
   Program11.RevOverContrast := 1;
   Program11.RopeEndCycle := 16#02;
   Program11.Spare4 := 16#01;
   Program11.RopeTime := 1500;
   Program11.RevOverClamp := 1;
   Program11.FilmForceFinalRev := 10;
   Program11.FilmPrestretchFinalRev := 100;
   Program11.ArmSpeed := 100;
   Program11.CarriageDown4Top := 500;
   Program11.TopDownTime := 1500;
   Program11.LapsUnderTop := 0;
   Program11.Spare6 := 0;
   Program11.Spare7 := 0;
   Program11.Spare8 := 0;
   Program11.Spare9 := 0;
   Program11.Spare10 := 0;
   Program11.Spare11 := 0;
   Program11.Spare12 := 0;
   Program11.Overlap0_1 := 0;
   Program11.Height1 := 130;
   Program11.Landmark1 := FALSE;
   Program11.Lifter1 := FALSE;
   Program11.SpareBit1H1 := FALSE;
   Program11.Airblower1 := TRUE;
   Program11.NextStep1 := TRUE;
   Program11.PressureP1 := TRUE;
   Program11.SpareByte2H1 := 16#00;
   Program11.Revolution1 := 1;
   Program11.RopeUnit1_1 := 16#01;
   Program11.RopeUnit1_2 := 16#01;
   Program11.FilmForce1 := 5;
   Program11.FilmPrestretch1 := 200;
   Program11.Spare3H1 := 0;
   Program11.Spare49 := 0;
   Program11.Spare50 := 0;
   Program11.Spare51 := 0;
   Program11.Spare52 := 0;
   Program11.Spare53 := 0;
   Program11.Overlap1_2 := 0;
   Program11.Height2 := 50;
   Program11.Landmark2 := FALSE;
   Program11.Lifter2 := FALSE;
   Program11.SpareBit1H2 := FALSE;
   Program11.Airblower2 := TRUE;
   Program11.NextStep2 := TRUE;
   Program11.PressureP2 := TRUE;
   Program11.SpareByte2H2 := 16#00;
   Program11.Revolution2 := 1;
   Program11.RopeUnit2_1 := 16#01;
   Program11.RopeUnit2_2 := 16#01;
   Program11.FilmForce2 := 20;
   Program11.FilmPrestretch2 := 200;
   Program11.Spare3H2 := 0;
   Program11.Spare54 := 0;
   Program11.Spare55 := 0;
   Program11.Spare56 := 0;
   Program11.Spare57 := 0;
   Program11.Spare58 := 0;
   Program11.Overlap2_3 := 100;
   Program11.Height3 := -50;
   Program11.Landmark3 := TRUE;
   Program11.Lifter3 := FALSE;
   Program11.SpareBit1H3 := FALSE;
   Program11.Airblower3 := TRUE;
   Program11.NextStep3 := TRUE;
   Program11.PressureP3 := TRUE;
   Program11.SpareByte2H3 := 16#00;
   Program11.Revolution3 := 2;
   Program11.RopeUnit3_1 := 16#01;
   Program11.RopeUnit3_2 := 16#01;
   Program11.FilmForce3 := 30;
   Program11.FilmPrestretch3 := 200;
   Program11.Spare3H3 := 0;
   Program11.Spare59 := 0;
   Program11.Spare60 := 0;
   Program11.Spare61 := 380;
   Program11.Spare62 := 2800;
   Program11.Spare63 := 0;
   Program11.Overlap3_4 := 100;
   Program11.Height4 := 100;
   Program11.Landmark4 := FALSE;
   Program11.Lifter4 := FALSE;
   Program11.SpareBit1H4 := FALSE;
   Program11.Airblower4 := TRUE;
   Program11.NextStep4 := TRUE;
   Program11.PressureP4 := TRUE;
   Program11.SpareByte2H4 := 16#00;
   Program11.Revolution4 := 3;
   Program11.RopeUnit4_1 := 16#02;
   Program11.RopeUnit4_2 := 16#02;
   Program11.FilmForce4 := 30;
   Program11.FilmPrestretch4 := 200;
   Program11.Spare3H4 := 0;
   Program11.Spare64 := 0;
   Program11.Spare65 := 0;
   Program11.Spare66 := 0;
   Program11.Spare67 := 0;
   Program11.Spare68 := 0;
   Program11.Overlap4_5 := 0;
   Program11.Height5 := 50;
   Program11.Landmark5 := FALSE;
   Program11.Lifter5 := FALSE;
   Program11.SpareBit1H5 := FALSE;
   Program11.Airblower5 := TRUE;
   Program11.NextStep5 := FALSE;
   Program11.PressureP5 := FALSE;
   Program11.SpareByte2H5 := 16#00;
   Program11.Revolution5 := 1;
   Program11.RopeUnit5_1 := 16#01;
   Program11.RopeUnit5_2 := 16#01;
   Program11.FilmForce5 := 30;
   Program11.FilmPrestretch5 := 200;
   Program11.Spare3H5 := 0;
   Program11.Spare69 := 0;
   Program11.Spare70 := 0;
   Program11.Spare71 := 0;
   Program11.Spare72 := 0;
   Program11.Spare73 := 0;
   Program11.Overlap5_6 := 100;
   Program11.Height6 := 50;
   Program11.Landmark6 := FALSE;
   Program11.Lifter6 := FALSE;
   Program11.SpareBit1H6 := FALSE;
   Program11.Airblower6 := TRUE;
   Program11.NextStep6 := FALSE;
   Program11.PressureP6 := FALSE;
   Program11.SpareByte2H6 := 16#00;
   Program11.Revolution6 := 2;
   Program11.RopeUnit6_1 := 16#02;
   Program11.RopeUnit6_2 := 16#01;
   Program11.FilmForce6 := 20;
   Program11.FilmPrestretch6 := 200;
   Program11.Spare3H6 := 0;
   Program11.Spare74 := 0;
   Program11.Spare75 := 0;
   Program11.Spare76 := 0;
   Program11.Spare77 := 0;
   Program11.Spare78 := 0;
   Program11.Overlap6_7 := 0;
   Program11.Height7 := 0;
   Program11.Landmark7 := FALSE;
   Program11.Lifter7 := FALSE;
   Program11.SpareBit1H7 := FALSE;
   Program11.Airblower7 := FALSE;
   Program11.NextStep7 := TRUE;
   Program11.PressureP7 := FALSE;
   Program11.SpareByte2H7 := 16#00;
   Program11.Revolution7 := 1;
   Program11.RopeUnit7_1 := 16#01;
   Program11.RopeUnit7_2 := 16#01;
   Program11.FilmForce7 := 0;
   Program11.FilmPrestretch7 := 100;
   Program11.Spare3H7 := 0;
   Program11.Spare79 := 0;
   Program11.Spare80 := 0;
   Program11.Spare81 := 0;
   Program11.Spare82 := 0;
   Program11.Spare83 := 0;
   Program11.Overlap7_8 := 0;
   Program11.Height8 := 0;
   Program11.Landmark8 := FALSE;
   Program11.Lifter8 := FALSE;
   Program11.SpareBit1H8 := FALSE;
   Program11.Airblower8 := FALSE;
   Program11.NextStep8 := TRUE;
   Program11.PressureP8 := FALSE;
   Program11.SpareByte2H8 := 16#00;
   Program11.Revolution8 := 1;
   Program11.RopeUnit8_1 := 16#01;
   Program11.RopeUnit8_2 := 16#01;
   Program11.FilmForce8 := 0;
   Program11.FilmPrestretch8 := 100;
   Program11.Spare3H8 := 0;
   Program11.Spare84 := 0;
   Program11.Spare85 := 0;
   Program11.Spare86 := 0;
   Program11.Spare87 := 0;
   Program11.Spare88 := 0;
   Program11.Overlap8_9 := 0;
   Program11.Height9 := 0;
   Program11.Landmark9 := FALSE;
   Program11.Lifter9 := FALSE;
   Program11.SpareBit1H9 := FALSE;
   Program11.Airblower9 := FALSE;
   Program11.NextStep9 := TRUE;
   Program11.PressureP9 := FALSE;
   Program11.SpareByte2H9 := 16#00;
   Program11.Revolution9 := 1;
   Program11.RopeUnit9_1 := 16#01;
   Program11.RopeUnit9_2 := 16#01;
   Program11.FilmForce9 := 0;
   Program11.FilmPrestretch9 := 100;
   Program11.Spare3H9 := 0;
   Program11.Spare89 := 0;
   Program11.Spare90 := 0;
   Program11.Spare91 := 0;
   Program11.Spare92 := 0;
   Program11.Spare93 := 0;
   Program11.Overlap9_10 := 0;
   Program11.Height10 := 0;
   Program11.Landmark10 := FALSE;
   Program11.Lifter10 := FALSE;
   Program11.SpareBit1H10 := FALSE;
   Program11.Airblower10 := FALSE;
   Program11.NextStep10 := FALSE;
   Program11.PressureP10 := FALSE;
   Program11.SpareByte2H10 := 16#00;
   Program11.Revolution10 := 1;
   Program11.RopeUnit10_1 := 16#01;
   Program11.RopeUnit10_2 := 16#01;
   Program11.FilmForce10 := 0;
   Program11.FilmPrestretch10 := 100;
   Program11.Spare3H10 := 0;
   Program11.Spare94 := 0;
   Program11.Spare95 := 0;
   Program11.Spare96 := 0;
   Program11.Spare97 := 0;
   Program11.Spare98 := 0;
   Program11.Overlap10_11 := 0;
   Program11.Height11 := 0;
   Program11.Landmark11 := FALSE;
   Program11.Lifter11 := FALSE;
   Program11.SpareBit1H11 := FALSE;
   Program11.Airblower11 := FALSE;
   Program11.NextStep11 := TRUE;
   Program11.PressureP11 := FALSE;
   Program11.SpareByte2H11 := 16#00;
   Program11.Revolution11 := 1;
   Program11.RopeUnit11_1 := 16#01;
   Program11.RopeUnit11_2 := 16#01;
   Program11.FilmForce11 := 0;
   Program11.FilmPrestretch11 := 100;
   Program11.Spare3H11 := 0;
   Program11.Spare99 := 0;
   Program11.Spare100 := 0;
   Program11.Spare101 := 0;
   Program11.Spare102 := 0;
   Program11.Spare103 := 0;
   Program11.Overlap11_12 := 0;
   Program11.Height12 := 0;
   Program11.Landmark12 := FALSE;
   Program11.Lifter12 := FALSE;
   Program11.SpareBit1H12 := FALSE;
   Program11.Airblower12 := FALSE;
   Program11.NextStep12 := FALSE;
   Program11.PressureP12 := FALSE;
   Program11.SpareByte2H12 := 16#00;
   Program11.Revolution12 := 1;
   Program11.RopeUnit12_1 := 16#01;
   Program11.RopeUnit12_2 := 16#01;
   Program11.FilmForce12 := 0;
   Program11.FilmPrestretch12 := 100;
   Program11.Spare3H12 := 0;
   Program11.Spare104 := 0;
   Program11.Spare105 := 0;
   Program11.Spare106 := 0;
   Program11.Spare107 := 0;
   Program11.Spare108 := 0;
END_DATA_BLOCK

